LIN {X 0,Y 390.078,Z 257.397,A -85,B 0,C 180,E1 -11718.916,E2 -11718.916} C_VEL
LIN {X 0,Y 390.01,Z 257.402,A -85,B 0,C 180,E1 -11722.228,E2 -11722.228} C_VEL
LIN {X 0,Y 390.089,Z 257.39,A -85,B 0,C 180,E1 -11725.737,E2 -11725.737} C_VEL
LIN {X 0,Y 390.02,Z 257.4,A -85,B 0,C 180,E1 -11729.104,E2 -11729.104} C_VEL
LIN {X 0,Y 390.006,Z 257.404,A -85,B 0,C 180,E1 -11732.716,E2 -11732.716} C_VEL
LIN {X 0,Y 390.018,Z 257.4,A -85,B 0,C 180,E1 -11735.819,E2 -11735.819} C_VEL
LIN {X 0,Y 390.032,Z 257.397,A -85,B 0,C 180,E1 -11739.213,E2 -11739.213} C_VEL
LIN {X 0,Y 390.078,Z 257.396,A -85,B 0,C 180,E1 -11742.381,E2 -11742.381} C_VEL
LIN {X 0,Y 390.074,Z 257.392,A -85,B 0,C 180,E1 -11745.36,E2 -11745.36} C_VEL
LIN {X 0,Y 390.056,Z 257.399,A -85,B 0,C 180,E1 -11748.191,E2 -11748.191} C_VEL
LIN {X 0,Y 390.045,Z 257.396,A -85,B 0,C 180,E1 -11750.903,E2 -11750.903} C_VEL
LIN {X 0,Y 390.032,Z 257.397,A -85,B 0,C 180,E1 -11754.789,E2 -11754.789} C_VEL
LIN {X 0,Y 389.97,Z 257.405,A -85,B 0,C 180,E1 -11758.492,E2 -11758.492} C_VEL
LIN {X 0,Y 390.061,Z 257.396,A -85,B 0,C 180,E1 -11762.066,E2 -11762.066} C_VEL
LIN {X 0,Y 390.027,Z 257.404,A -85,B 0,C 180,E1 -11765.516,E2 -11765.516} C_VEL
LIN {X 0,Y 390.049,Z 257.396,A -85,B 0,C 180,E1 -11768.878,E2 -11768.878} C_VEL
LIN {X 0,Y 390.088,Z 257.395,A -85,B 0,C 180,E1 -11772.689,E2 -11772.689} C_VEL
LIN {X 0,Y 390.132,Z 257.39,A -85,B 0,C 180,E1 -11776.56,E2 -11776.56} C_VEL
LIN {X 0,Y 390.118,Z 257.391,A -85,B 0,C 180,E1 -11779.622,E2 -11779.622} C_VEL
LIN {X 0,Y 390.303,Z 257.447,A -85,B 0,C 180,E1 -11782.673,E2 -11782.673} C_VEL
LIN {X 0,Y 390.823,Z 259.339,A -85,B 0,C 180,E1 -11783.093,E2 -11783.093} C_VEL
LIN {X 0,Y 392.36,Z 261.617,A -85,B 0,C 180,E1 -11784.217,E2 -11784.217} C_VEL
LIN {X 0,Y 394.306,Z 263.039,A -85,B 0,C 180,E1 -11785.912,E2 -11785.912} C_VEL
LIN {X 0,Y 395.192,Z 263.267,A -85,B 0,C 180,E1 -11786.942,E2 -11786.942} C_VEL
LIN {X 0,Y 396.203,Z 263.5,A -85,B 0,C 180,E1 -11788.984,E2 -11788.984} C_VEL
LIN {X 0,Y 396.371,Z 263.477,A -85,B 0,C 180,E1 -11790,E2 -11790} C_VEL
LIN {X 0,Y 395.805,Z 263.406,A -85,B 0,C 180,E1 -11792.035,E2 -11792.035} C_VEL
LIN {X 0,Y 394.435,Z 263.067,A -85,B 0,C 180,E1 -11793.94,E2 -11793.94} C_VEL
LIN {X 0,Y 392.534,Z 261.798,A -85,B 0,C 180,E1 -11795.651,E2 -11795.651} C_VEL
LIN {X 0,Y 390.904,Z 259.538,A -85,B 0,C 180,E1 -11796.841,E2 -11796.841} C_VEL
LIN {X 0,Y 390.334,Z 257.663,A -85,B 0,C 180,E1 -11797.298,E2 -11797.298} C_VEL
LIN {X 0,Y 390.276,Z 257.373,A -85,B 0,C 180,E1 -11797.472,E2 -11797.472} C_VEL
LIN {X 0,Y 390.097,Z 257.393,A -85,B 0,C 180,E1 -11801.43,E2 -11801.43} C_VEL
LIN {X 0,Y 390.089,Z 257.397,A -85,B 0,C 180,E1 -11804.609,E2 -11804.609} C_VEL
LIN {X 0,Y 390.07,Z 257.397,A -85,B 0,C 180,E1 -11807.836,E2 -11807.836} C_VEL
LIN {X 0,Y 390.049,Z 257.396,A -85,B 0,C 180,E1 -11811.122,E2 -11811.122} C_VEL
LIN {X 0,Y 390.027,Z 257.404,A -85,B 0,C 180,E1 -11814.484,E2 -11814.484} C_VEL
LIN {X 0,Y 390.059,Z 257.397,A -85,B 0,C 180,E1 -11818.029,E2 -11818.029} C_VEL
LIN {X 0,Y 389.96,Z 257.408,A -85,B 0,C 180,E1 -11820.785,E2 -11820.785} C_VEL
LIN {X 0,Y 389.284,Z 257.493,A -85,B 0,C 180,E1 -11821.647,E2 -11821.647} C_VEL
LIN {X 0,Y 386.437,Z 257.845,A -85,B 0,C 180,E1 -11823.049,E2 -11823.049} C_VEL
LIN {X 0,Y 384.041,Z 258.15,A -85,B 0,C 180,E1 -11824.182,E2 -11824.182} C_VEL
LIN {X 0,Y 383.023,Z 258.271,A -85,B 0,C 180,E1 -11825.058,E2 -11825.058} C_VEL
LIN {X 0,Y 382.945,Z 258.28,A -85,B 0,C 180,E1 -11825.355,E2 -11825.355} C_VEL
LIN {X 0,Y 382.958,Z 258.28,A -85,B 0,C 180,E1 -11828.605,E2 -11828.605} C_VEL
LIN {X 0,Y 382.998,Z 258.274,A -85,B 0,C 180,E1 -11831.344,E2 -11831.344} C_VEL
LIN {X 0,Y 383.025,Z 258.272,A -85,B 0,C 180,E1 -11834.32,E2 -11834.32} C_VEL
LIN {X 0,Y 383.032,Z 258.271,A -85,B 0,C 180,E1 -11837.255,E2 -11837.255} C_VEL
LIN {X 0,Y 382.98,Z 258.276,A -85,B 0,C 180,E1 -11840.418,E2 -11840.418} C_VEL
LIN {X 0,Y 382.987,Z 258.277,A -85,B 0,C 180,E1 -11844.051,E2 -11844.051} C_VEL
LIN {X 0,Y 382.968,Z 258.284,A -85,B 0,C 180,E1 -11847.58,E2 -11847.58} C_VEL
LIN {X 0,Y 382.955,Z 258.279,A -85,B 0,C 180,E1 -11850.306,E2 -11850.306} C_VEL
LIN {X 0,Y 383.05,Z 258.268,A -85,B 0,C 180,E1 -11854.027,E2 -11854.027} C_VEL
LIN {X 0,Y 382.964,Z 258.284,A -85,B 0,C 180,E1 -11857.341,E2 -11857.341} C_VEL
LIN {X 0,Y 383.033,Z 258.271,A -85,B 0,C 180,E1 -11860.723,E2 -11860.723} C_VEL
LIN {X 0,Y 383.058,Z 258.266,A -85,B 0,C 180,E1 -11864.033,E2 -11864.033} C_VEL
LIN {X 0,Y 383.117,Z 258.263,A -85,B 0,C 180,E1 -11867.29,E2 -11867.29} C_VEL
LIN {X 0,Y 383.126,Z 258.259,A -85,B 0,C 180,E1 -11870.504,E2 -11870.504} C_VEL
LIN {X 0,Y 383.246,Z 258.243,A -85,B 0,C 180,E1 -11873.69,E2 -11873.69} C_VEL
LIN {X 0,Y 383.373,Z 258.227,A -85,B 0,C 180,E1 -11877.905,E2 -11877.905} C_VEL
LIN {X 0,Y 383.505,Z 258.211,A -85,B 0,C 180,E1 -11880.006,E2 -11880.006} C_VEL
LIN {X 0,Y 383.196,Z 258.251,A -85,B 0,C 180,E1 -11883.16,E2 -11883.16} C_VEL
LIN {X 0,Y 383.254,Z 258.245,A -85,B 0,C 180,E1 -11886.323,E2 -11886.323} C_VEL
LIN {X 0,Y 383.138,Z 258.256,A -85,B 0,C 180,E1 -11889.508,E2 -11889.508} C_VEL
LIN {X 0,Y 383.125,Z 258.258,A -85,B 0,C 180,E1 -11893.541,E2 -11893.541} C_VEL
LIN {X 0,Y 383.095,Z 258.262,A -85,B 0,C 180,E1 -11897.074,E2 -11897.074} C_VEL
LIN {X 0,Y 383.032,Z 258.272,A -85,B 0,C 180,E1 -11900.651,E2 -11900.651} C_VEL
LIN {X 0,Y 383.018,Z 258.274,A -85,B 0,C 180,E1 -11903.813,E2 -11903.813} C_VEL
LIN {X 0,Y 382.993,Z 258.274,A -85,B 0,C 180,E1 -11907.312,E2 -11907.312} C_VEL
LIN {X 0,Y 382.988,Z 258.275,A -85,B 0,C 180,E1 -11910.923,E2 -11910.923} C_VEL
LIN {X 0,Y 383.02,Z 258.274,A -85,B 0,C 180,E1 -11914.673,E2 -11914.673} C_VEL
LIN {X 0,Y 383.006,Z 258.279,A -85,B 0,C 180,E1 -11917.907,E2 -11917.907} C_VEL
LIN {X 0,Y 383.421,Z 261.152,A -85,B 0,C 180,E1 -11921.295,E2 -11921.295} C_VEL
LIN {X 0,Y 383.824,Z 264.04,A -85,B 0,C 180,E1 -11924.431,E2 -11924.431} C_VEL
LIN {X 0,Y 384.033,Z 267.009,A -85,B 0,C 180,E1 -11927.382,E2 -11927.382} C_VEL
LIN {X 0,Y 383.857,Z 270.176,A -85,B 0,C 180,E1 -11930.267,E2 -11930.267} C_VEL
LIN {X 0,Y 383.506,Z 274.24,A -85,B 0,C 180,E1 -11933.744,E2 -11933.744} C_VEL
LIN {X 0,Y 383.169,Z 277.795,A -85,B 0,C 180,E1 -11936.617,E2 -11936.617} C_VEL
LIN {X 0,Y 382.7,Z 282.543,A -85,B 0,C 180,E1 -11940.276,E2 -11940.276} C_VEL
LIN {X 0,Y 382.294,Z 287.36,A -85,B 0,C 180,E1 -11943.82,E2 -11943.82} C_VEL
LIN {X 0,Y 382.041,Z 292.216,A -85,B 0,C 180,E1 -11947.275,E2 -11947.275} C_VEL
LIN {X 0,Y 381.798,Z 297.479,A -85,B 0,C 180,E1 -11950.93,E2 -11950.93} C_VEL
LIN {X 0,Y 381.775,Z 297.832,A -85,B 0,C 180,E1 -11951.103,E2 -11951.103} C_VEL
LIN {X 0,Y 383.933,Z 308.212,A -85,B 0,C 180,E1 -11951.559,E2 -11951.559} C_VEL
LIN {X 0,Y 385.499,Z 317.173,A -85,B 0,C 180,E1 -11952.051,E2 -11952.051} C_VEL
LIN {X 0,Y 386.76,Z 326.079,A -85,B 0,C 180,E1 -11952.634,E2 -11952.634} C_VEL
LIN {X 0,Y 387.065,Z 332.785,A -85,B 0,C 180,E1 -11953.112,E2 -11953.112} C_VEL
LIN {X 0,Y 386.15,Z 343.695,A -85,B 0,C 180,E1 -11954.022,E2 -11954.022} C_VEL
LIN {X 0,Y 385.323,Z 352.64,A -85,B 0,C 180,E1 -11954.936,E2 -11954.936} C_VEL
LIN {X 0,Y 384.651,Z 360.342,A -85,B 0,C 180,E1 -11955.874,E2 -11955.874} C_VEL
LIN {X 0,Y 383.975,Z 368.393,A -85,B 0,C 180,E1 -11957.044,E2 -11957.044} C_VEL
LIN {X 0,Y 383.342,Z 374.594,A -85,B 0,C 180,E1 -11958.098,E2 -11958.098} C_VEL
LIN {X 0,Y 382.751,Z 381.132,A -85,B 0,C 180,E1 -11959.42,E2 -11959.42} C_VEL
LIN {X 0,Y 382.377,Z 385.634,A -85,B 0,C 180,E1 -11960.479,E2 -11960.479} C_VEL
LIN {X 0,Y 381.964,Z 391.125,A -85,B 0,C 180,E1 -11962.068,E2 -11962.068} C_VEL
LIN {X 0,Y 381.726,Z 395.45,A -85,B 0,C 180,E1 -11963.658,E2 -11963.658} C_VEL
LIN {X 0,Y 381.65,Z 397.817,A -85,B 0,C 180,E1 -11964.717,E2 -11964.717} C_VEL
LIN {X 0,Y 381.624,Z 399.616,A -85,B 0,C 180,E1 -11965.776,E2 -11965.776} C_VEL
LIN {X 0,Y 381.563,Z 402.06,A -85,B 0,C 180,E1 -11967.889,E2 -11967.889} C_VEL
LIN {X 0,Y 381.598,Z 402.649,A -85,B 0,C 180,E1 -11968.945,E2 -11968.945} C_VEL
LIN {X 0,Y 381.598,Z 402.649,A -85,B 0,C 180,E1 -11971.055,E2 -11971.055} C_VEL
LIN {X 0,Y 381.563,Z 402.06,A -85,B 0,C 180,E1 -11972.111,E2 -11972.111} C_VEL
LIN {X 0,Y 381.624,Z 399.616,A -85,B 0,C 180,E1 -11974.224,E2 -11974.224} C_VEL
LIN {X 0,Y 381.65,Z 397.817,A -85,B 0,C 180,E1 -11975.283,E2 -11975.283} C_VEL
LIN {X 0,Y 381.795,Z 394.21,A -85,B 0,C 180,E1 -11976.872,E2 -11976.872} C_VEL
LIN {X 0,Y 382.075,Z 389.465,A -85,B 0,C 180,E1 -11978.462,E2 -11978.462} C_VEL
LIN {X 0,Y 382.544,Z 383.443,A -85,B 0,C 180,E1 -11980.051,E2 -11980.051} C_VEL
LIN {X 0,Y 383.071,Z 377.346,A -85,B 0,C 180,E1 -11981.374,E2 -11981.374} C_VEL
LIN {X 0,Y 383.641,Z 371.646,A -85,B 0,C 180,E1 -11982.43,E2 -11982.43} C_VEL
LIN {X 0,Y 384.394,Z 363.091,A -85,B 0,C 180,E1 -11983.749,E2 -11983.749} C_VEL
LIN {X 0,Y 385.11,Z 354.909,A -85,B 0,C 180,E1 -11984.802,E2 -11984.802} C_VEL
LIN {X 0,Y 385.872,Z 346.398,A -85,B 0,C 180,E1 -11985.719,E2 -11985.719} C_VEL
LIN {X 0,Y 386.581,Z 337.681,A -85,B 0,C 180,E1 -11986.502,E2 -11986.502} C_VEL
LIN {X 0,Y 387.137,Z 330.218,A -85,B 0,C 180,E1 -11987.07,E2 -11987.07} C_VEL
LIN {X 0,Y 386.004,Z 320.346,A -85,B 0,C 180,E1 -11987.757,E2 -11987.757} C_VEL
LIN {X 0,Y 384.122,Z 309.199,A -85,B 0,C 180,E1 -11988.392,E2 -11988.392} C_VEL
LIN {X 0,Y 381.847,Z 298.335,A -85,B 0,C 180,E1 -11988.88,E2 -11988.88} C_VEL
LIN {X 0,Y 381.777,Z 297.67,A -85,B 0,C 180,E1 -11988.932,E2 -11988.932} C_VEL
LIN {X 0,Y 382.043,Z 292.21,A -85,B 0,C 180,E1 -11992.725,E2 -11992.725} C_VEL
LIN {X 0,Y 382.294,Z 287.352,A -85,B 0,C 180,E1 -11996.18,E2 -11996.18} C_VEL
LIN {X 0,Y 382.701,Z 282.543,A -85,B 0,C 180,E1 -11999.724,E2 -11999.724} C_VEL
LIN {X 0,Y 383.07,Z 278.991,A -85,B 0,C 180,E1 -12002.436,E2 -12002.436} C_VEL
LIN {X 0,Y 383.457,Z 274.66,A -85,B 0,C 180,E1 -12005.908,E2 -12005.908} C_VEL
LIN {X 0,Y 383.718,Z 271.563,A -85,B 0,C 180,E1 -12008.514,E2 -12008.514} C_VEL
LIN {X 0,Y 383.974,Z 268.349,A -85,B 0,C 180,E1 -12011.367,E2 -12011.367} C_VEL
LIN {X 0,Y 383.99,Z 265.506,A -85,B 0,C 180,E1 -12014.066,E2 -12014.066} C_VEL
LIN {X 0,Y 383.565,Z 262.396,A -85,B 0,C 180,E1 -12017.312,E2 -12017.312} C_VEL
LIN {X 0,Y 383.222,Z 259.706,A -85,B 0,C 180,E1 -12020.374,E2 -12020.374} C_VEL
LIN {X 0,Y 383.007,Z 258.279,A -85,B 0,C 180,E1 -12022.093,E2 -12022.093} C_VEL
LIN {X 0,Y 383.025,Z 258.277,A -85,B 0,C 180,E1 -12025.328,E2 -12025.328} C_VEL
LIN {X 0,Y 382.988,Z 258.275,A -85,B 0,C 180,E1 -12029.077,E2 -12029.077} C_VEL
LIN {X 0,Y 382.993,Z 258.274,A -85,B 0,C 180,E1 -12032.688,E2 -12032.688} C_VEL
LIN {X 0,Y 383.018,Z 258.274,A -85,B 0,C 180,E1 -12036.187,E2 -12036.187} C_VEL
LIN {X 0,Y 383.058,Z 258.271,A -85,B 0,C 180,E1 -12039.593,E2 -12039.593} C_VEL
LIN {X 0,Y 383.095,Z 258.262,A -85,B 0,C 180,E1 -12042.926,E2 -12042.926} C_VEL
LIN {X 0,Y 383.125,Z 258.258,A -85,B 0,C 180,E1 -12046.459,E2 -12046.459} C_VEL
LIN {X 0,Y 383.138,Z 258.256,A -85,B 0,C 180,E1 -12050.492,E2 -12050.492} C_VEL
LIN {X 0,Y 383.254,Z 258.245,A -85,B 0,C 180,E1 -12053.677,E2 -12053.677} C_VEL
LIN {X 0,Y 383.366,Z 258.229,A -85,B 0,C 180,E1 -12057.893,E2 -12057.893} C_VEL
LIN {X 0,Y 383.505,Z 258.211,A -85,B 0,C 180,E1 -12059.994,E2 -12059.994} C_VEL
LIN {X 0,Y 383.23,Z 258.251,A -85,B 0,C 180,E1 -12063.147,E2 -12063.147} C_VEL
LIN {X 0,Y 383.225,Z 258.245,A -85,B 0,C 180,E1 -12066.59,E2 -12066.59} C_VEL
LIN {X 0,Y 383.126,Z 258.259,A -85,B 0,C 180,E1 -12069.496,E2 -12069.496} C_VEL
LIN {X 0,Y 383.106,Z 258.261,A -85,B 0,C 180,E1 -12073.53,E2 -12073.53} C_VEL
LIN {X 0,Y 383.071,Z 258.268,A -85,B 0,C 180,E1 -12077.063,E2 -12077.063} C_VEL
LIN {X 0,Y 383.003,Z 258.279,A -85,B 0,C 180,E1 -12080.64,E2 -12080.64} C_VEL
LIN {X 0,Y 382.994,Z 258.274,A -85,B 0,C 180,E1 -12083.802,E2 -12083.802} C_VEL
LIN {X 0,Y 383.049,Z 258.269,A -85,B 0,C 180,E1 -12086.117,E2 -12086.117} C_VEL
LIN {X 0,Y 382.955,Z 258.279,A -85,B 0,C 180,E1 -12089.694,E2 -12089.694} C_VEL
LIN {X 0,Y 382.966,Z 258.277,A -85,B 0,C 180,E1 -12093.395,E2 -12093.395} C_VEL
LIN {X 0,Y 382.994,Z 258.279,A -85,B 0,C 180,E1 -12096.159,E2 -12096.159} C_VEL
LIN {X 0,Y 382.978,Z 258.279,A -85,B 0,C 180,E1 -12099.951,E2 -12099.951} C_VEL
LIN {X 0,Y 383.022,Z 258.272,A -85,B 0,C 180,E1 -12102.783,E2 -12102.783} C_VEL
LIN {X 0,Y 383.027,Z 258.273,A -85,B 0,C 180,E1 -12105.795,E2 -12105.795} C_VEL
LIN {X 0,Y 382.996,Z 258.274,A -85,B 0,C 180,E1 -12108.781,E2 -12108.781} C_VEL
LIN {X 0,Y 382.952,Z 258.284,A -85,B 0,C 180,E1 -12112.091,E2 -12112.091} C_VEL
LIN {X 0,Y 382.965,Z 258.279,A -85,B 0,C 180,E1 -12115.328,E2 -12115.328} C_VEL
LIN {X 0,Y 382.93,Z 258.283,A -85,B 0,C 180,E1 -12119.078,E2 -12119.078} C_VEL
LIN {X 0,Y 382.999,Z 258.273,A -85,B 0,C 180,E1 -12122.694,E2 -12122.694} C_VEL
LIN {X 0,Y 382.99,Z 258.276,A -85,B 0,C 180,E1 -12126.19,E2 -12126.19} C_VEL
LIN {X 0,Y 383.022,Z 258.277,A -85,B 0,C 180,E1 -12129.597,E2 -12129.597} C_VEL
LIN {X 0,Y 383.045,Z 258.273,A -85,B 0,C 180,E1 -12132.929,E2 -12132.929} C_VEL
LIN {X 0,Y 383.063,Z 258.27,A -85,B 0,C 180,E1 -12136.462,E2 -12136.462} C_VEL
LIN {X 0,Y 383.112,Z 258.454,A -85,B 0,C 180,E1 -12139.597,E2 -12139.597} C_VEL
LIN {X 0,Y 383.731,Z 260.437,A -85,B 0,C 180,E1 -12139.914,E2 -12139.914} C_VEL
LIN {X 0,Y 385.194,Z 262.473,A -85,B 0,C 180,E1 -12140.615,E2 -12140.615} C_VEL
LIN {X 0,Y 387.433,Z 263.895,A -85,B 0,C 180,E1 -12141.656,E2 -12141.656} C_VEL
LIN {X 0,Y 388.819,Z 264.578,A -85,B 0,C 180,E1 -12142.393,E2 -12142.393} C_VEL
LIN {X 0,Y 389.954,Z 266.887,A -85,B 0,C 180,E1 -12143.142,E2 -12143.142} C_VEL
LIN {X 0,Y 391.787,Z 269.021,A -85,B 0,C 180,E1 -12144.467,E2 -12144.467} C_VEL
LIN {X 0,Y 393.419,Z 270.082,A -85,B 0,C 180,E1 -12145.903,E2 -12145.903} C_VEL
LIN {X 0,Y 394.315,Z 270.311,A -85,B 0,C 180,E1 -12146.935,E2 -12146.935} C_VEL
LIN {X 0,Y 395.344,Z 270.547,A -85,B 0,C 180,E1 -12148.981,E2 -12148.981} C_VEL
LIN {X 0,Y 395.505,Z 270.523,A -85,B 0,C 180,E1 -12150,E2 -12150} C_VEL
LIN {X 0,Y 394.942,Z 270.452,A -85,B 0,C 180,E1 -12152.04,E2 -12152.04} C_VEL
LIN {X 0,Y 393.419,Z 270.083,A -85,B 0,C 180,E1 -12154.097,E2 -12154.097} C_VEL
LIN {X 0,Y 391.44,Z 268.741,A -85,B 0,C 180,E1 -12155.796,E2 -12155.796} C_VEL
LIN {X 0,Y 389.612,Z 266.328,A -85,B 0,C 180,E1 -12157.089,E2 -12157.089} C_VEL
LIN {X 0,Y 388.598,Z 264.268,A -85,B 0,C 180,E1 -12157.735,E2 -12157.735} C_VEL
LIN {X 0,Y 386.111,Z 263.175,A -85,B 0,C 180,E1 -12158.966,E2 -12158.966} C_VEL
LIN {X 0,Y 384.201,Z 261.296,A -85,B 0,C 180,E1 -12159.861,E2 -12159.861} C_VEL
LIN {X 0,Y 383.293,Z 259.34,A -85,B 0,C 180,E1 -12160.298,E2 -12160.298} C_VEL
LIN {X 0,Y 383.073,Z 258.269,A -85,B 0,C 180,E1 -12160.438,E2 -12160.438} C_VEL
LIN {X 0,Y 383.066,Z 258.269,A -85,B 0,C 180,E1 -12163.798,E2 -12163.798} C_VEL
LIN {X 0,Y 383.035,Z 258.273,A -85,B 0,C 180,E1 -12167.458,E2 -12167.458} C_VEL
LIN {X 0,Y 383.004,Z 258.277,A -85,B 0,C 180,E1 -12170.664,E2 -12170.664} C_VEL
LIN {X 0,Y 382.99,Z 258.276,A -85,B 0,C 180,E1 -12173.81,E2 -12173.81} C_VEL
LIN {X 0,Y 382.999,Z 258.273,A -85,B 0,C 180,E1 -12177.306,E2 -12177.306} C_VEL
LIN {X 0,Y 382.93,Z 258.283,A -85,B 0,C 180,E1 -12180.922,E2 -12180.922} C_VEL
LIN {X 0,Y 382.965,Z 258.279,A -85,B 0,C 180,E1 -12184.672,E2 -12184.672} C_VEL
LIN {X 0,Y 382.945,Z 258.28,A -85,B 0,C 180,E1 -12185.355,E2 -12185.355} C_VEL
LIN {X 0,Y 382.302,Z 258.366,A -85,B 0,C 180,E1 -12186.233,E2 -12186.233} C_VEL
LIN {X 0,Y 379.489,Z 258.724,A -85,B 0,C 180,E1 -12187.661,E2 -12187.661} C_VEL
LIN {X 0,Y 377.087,Z 259.025,A -85,B 0,C 180,E1 -12188.816,E2 -12188.816} C_VEL
LIN {X 0,Y 376.041,Z 259.149,A -85,B 0,C 180,E1 -12189.708,E2 -12189.708} C_VEL
LIN {X 0,Y 375.949,Z 259.158,A -85,B 0,C 180,E1 -12190.01,E2 -12190.01} C_VEL
LIN {X 0,Y 375.955,Z 259.156,A -85,B 0,C 180,E1 -12193.761,E2 -12193.761} C_VEL
LIN {X 0,Y 375.955,Z 259.151,A -85,B 0,C 180,E1 -12196.806,E2 -12196.806} C_VEL
LIN {X 0,Y 375.957,Z 259.154,A -85,B 0,C 180,E1 -12200.034,E2 -12200.034} C_VEL
LIN {X 0,Y 375.926,Z 259.159,A -85,B 0,C 180,E1 -12203.501,E2 -12203.501} C_VEL
LIN {X 0,Y 375.923,Z 259.158,A -85,B 0,C 180,E1 -12205.895,E2 -12205.895} C_VEL
LIN {X 0,Y 375.929,Z 259.159,A -85,B 0,C 180,E1 -12209.694,E2 -12209.694} C_VEL
LIN {X 0,Y 375.989,Z 259.152,A -85,B 0,C 180,E1 -12213.354,E2 -12213.354} C_VEL
LIN {X 0,Y 375.951,Z 259.153,A -85,B 0,C 180,E1 -12216.894,E2 -12216.894} C_VEL
LIN {X 0,Y 375.971,Z 259.149,A -85,B 0,C 180,E1 -12220.346,E2 -12220.346} C_VEL
LIN {X 0,Y 376.003,Z 259.146,A -85,B 0,C 180,E1 -12223.725,E2 -12223.725} C_VEL
LIN {X 0,Y 376.084,Z 259.141,A -85,B 0,C 180,E1 -12227.049,E2 -12227.049} C_VEL
LIN {X 0,Y 376.096,Z 259.134,A -85,B 0,C 180,E1 -12230.325,E2 -12230.325} C_VEL
LIN {X 0,Y 376.205,Z 259.121,A -85,B 0,C 180,E1 -12233.571,E2 -12233.571} C_VEL
LIN {X 0,Y 376.339,Z 259.103,A -85,B 0,C 180,E1 -12237.866,E2 -12237.866} C_VEL
LIN {X 0,Y 376.474,Z 259.086,A -85,B 0,C 180,E1 -12240.006,E2 -12240.006} C_VEL
LIN {X 0,Y 376.331,Z 259.105,A -85,B 0,C 180,E1 -12242.147,E2 -12242.147} C_VEL
LIN {X 0,Y 376.213,Z 259.123,A -85,B 0,C 180,E1 -12246.441,E2 -12246.441} C_VEL
LIN {X 0,Y 376.109,Z 259.132,A -85,B 0,C 180,E1 -12249.687,E2 -12249.687} C_VEL
LIN {X 0,Y 376.089,Z 259.134,A -85,B 0,C 180,E1 -12253.663,E2 -12253.663} C_VEL
LIN {X 0,Y 376.034,Z 259.141,A -85,B 0,C 180,E1 -12257.405,E2 -12257.405} C_VEL
LIN {X 0,Y 375.982,Z 259.149,A -85,B 0,C 180,E1 -12260.837,E2 -12260.837} C_VEL
LIN {X 0,Y 375.967,Z 259.154,A -85,B 0,C 180,E1 -12264.289,E2 -12264.289} C_VEL
LIN {X 0,Y 375.937,Z 259.157,A -85,B 0,C 180,E1 -12267.869,E2 -12267.869} C_VEL
LIN {X 0,Y 375.964,Z 259.152,A -85,B 0,C 180,E1 -12271.567,E2 -12271.567} C_VEL
LIN {X 0,Y 375.958,Z 259.153,A -85,B 0,C 180,E1 -12275.421,E2 -12275.421} C_VEL
LIN {X 0,Y 375.958,Z 259.155,A -85,B 0,C 180,E1 -12276.746,E2 -12276.746} C_VEL
LIN {X 0,Y 376.032,Z 259.734,A -85,B 0,C 180,E1 -12278.283,E2 -12278.283} C_VEL
LIN {X 0,Y 376.457,Z 262.579,A -85,B 0,C 180,E1 -12281.692,E2 -12281.692} C_VEL
LIN {X 0,Y 376.875,Z 265.757,A -85,B 0,C 180,E1 -12285.129,E2 -12285.129} C_VEL
LIN {X 0,Y 376.966,Z 268.497,A -85,B 0,C 180,E1 -12287.844,E2 -12287.844} C_VEL
LIN {X 0,Y 376.776,Z 271.531,A -85,B 0,C 180,E1 -12290.64,E2 -12290.64} C_VEL
LIN {X 0,Y 376.488,Z 274.693,A -85,B 0,C 180,E1 -12293.394,E2 -12293.394} C_VEL
LIN {X 0,Y 376.039,Z 279.289,A -85,B 0,C 180,E1 -12297.181,E2 -12297.181} C_VEL
LIN {X 0,Y 375.738,Z 282.45,A -85,B 0,C 180,E1 -12299.668,E2 -12299.668} C_VEL
LIN {X 0,Y 375.267,Z 287.244,A -85,B 0,C 180,E1 -12303.291,E2 -12303.291} C_VEL
LIN {X 0,Y 375.003,Z 292.076,A -85,B 0,C 180,E1 -12306.824,E2 -12306.824} C_VEL
LIN {X 0,Y 374.753,Z 297.629,A -85,B 0,C 180,E1 -12310.735,E2 -12310.735} C_VEL
LIN {X 0,Y 376.778,Z 307.363,A -85,B 0,C 180,E1 -12311.17,E2 -12311.17} C_VEL
LIN {X 0,Y 378.522,Z 317.005,A -85,B 0,C 180,E1 -12311.711,E2 -12311.711} C_VEL
LIN {X 0,Y 379.834,Z 326.248,A -85,B 0,C 180,E1 -12312.333,E2 -12312.333} C_VEL
LIN {X 0,Y 380.262,Z 332.59,A -85,B 0,C 180,E1 -12312.8,E2 -12312.8} C_VEL
LIN {X 0,Y 379.323,Z 343.5,A -85,B 0,C 180,E1 -12313.726,E2 -12313.726} C_VEL
LIN {X 0,Y 378.437,Z 352.444,A -85,B 0,C 180,E1 -12314.655,E2 -12314.655} C_VEL
LIN {X 0,Y 377.712,Z 360.515,A -85,B 0,C 180,E1 -12315.662,E2 -12315.662} C_VEL
LIN {X 0,Y 377.039,Z 368.198,A -85,B 0,C 180,E1 -12316.801,E2 -12316.801} C_VEL
LIN {X 0,Y 376.386,Z 374.399,A -85,B 0,C 180,E1 -12317.874,E2 -12317.874} C_VEL
LIN {X 0,Y 375.73,Z 380.936,A -85,B 0,C 180,E1 -12319.22,E2 -12319.22} C_VEL
LIN {X 0,Y 375.336,Z 385.438,A -85,B 0,C 180,E1 -12320.298,E2 -12320.298} C_VEL
LIN {X 0,Y 374.901,Z 390.93,A -85,B 0,C 180,E1 -12321.918,E2 -12321.918} C_VEL
LIN {X 0,Y 374.647,Z 395.255,A -85,B 0,C 180,E1 -12323.538,E2 -12323.538} C_VEL
LIN {X 0,Y 374.561,Z 397.622,A -85,B 0,C 180,E1 -12324.617,E2 -12324.617} C_VEL
LIN {X 0,Y 374.53,Z 399.421,A -85,B 0,C 180,E1 -12325.695,E2 -12325.695} C_VEL
LIN {X 0,Y 374.462,Z 401.865,A -85,B 0,C 180,E1 -12327.849,E2 -12327.849} C_VEL
LIN {X 0,Y 374.499,Z 402.455,A -85,B 0,C 180,E1 -12328.925,E2 -12328.925} C_VEL
LIN {X 0,Y 374.499,Z 402.455,A -85,B 0,C 180,E1 -12331.075,E2 -12331.075} C_VEL
LIN {X 0,Y 374.462,Z 401.865,A -85,B 0,C 180,E1 -12332.151,E2 -12332.151} C_VEL
LIN {X 0,Y 374.53,Z 399.421,A -85,B 0,C 180,E1 -12334.305,E2 -12334.305} C_VEL
LIN {X 0,Y 374.595,Z 396.162,A -85,B 0,C 180,E1 -12336.06,E2 -12336.06} C_VEL
LIN {X 0,Y 374.812,Z 392.484,A -85,B 0,C 180,E1 -12337.542,E2 -12337.542} C_VEL
LIN {X 0,Y 375.175,Z 387.354,A -85,B 0,C 180,E1 -12339.162,E2 -12339.162} C_VEL
LIN {X 0,Y 375.65,Z 382.092,A -85,B 0,C 180,E1 -12340.51,E2 -12340.51} C_VEL
LIN {X 0,Y 376.217,Z 375.774,A -85,B 0,C 180,E1 -12341.858,E2 -12341.858} C_VEL
LIN {X 0,Y 376.877,Z 369.825,A -85,B 0,C 180,E1 -12342.931,E2 -12342.931} C_VEL
LIN {X 0,Y 377.62,Z 361.709,A -85,B 0,C 180,E1 -12344.171,E2 -12344.171} C_VEL
LIN {X 0,Y 378.421,Z 352.443,A -85,B 0,C 180,E1 -12345.346,E2 -12345.346} C_VEL
LIN {X 0,Y 379.385,Z 342.147,A -85,B 0,C 180,E1 -12346.409,E2 -12346.409} C_VEL
LIN {X 0,Y 380.288,Z 331.449,A -85,B 0,C 180,E1 -12347.288,E2 -12347.288} C_VEL
LIN {X 0,Y 379.081,Z 320.707,A -85,B 0,C 180,E1 -12348.062,E2 -12348.062} C_VEL
LIN {X 0,Y 377.189,Z 309.445,A -85,B 0,C 180,E1 -12348.725,E2 -12348.725} C_VEL
LIN {X 0,Y 374.81,Z 298.298,A -85,B 0,C 180,E1 -12349.244,E2 -12349.244} C_VEL
LIN {X 0,Y 374.752,Z 297.506,A -85,B 0,C 180,E1 -12349.3,E2 -12349.3} C_VEL
LIN {X 0,Y 375.016,Z 291.876,A -85,B 0,C 180,E1 -12353.316,E2 -12353.316} C_VEL
LIN {X 0,Y 375.266,Z 287.234,A -85,B 0,C 180,E1 -12356.709,E2 -12356.709} C_VEL
LIN {X 0,Y 375.763,Z 282.052,A -85,B 0,C 180,E1 -12360.638,E2 -12360.638} C_VEL
LIN {X 0,Y 376.182,Z 277.711,A -85,B 0,C 180,E1 -12364.088,E2 -12364.088} C_VEL
LIN {X 0,Y 376.494,Z 274.604,A -85,B 0,C 180,E1 -12366.679,E2 -12366.679} C_VEL
LIN {X 0,Y 376.831,Z 270.678,A -85,B 0,C 180,E1 -12370.118,E2 -12370.118} C_VEL
LIN {X 0,Y 377.005,Z 267.25,A -85,B 0,C 180,E1 -12373.357,E2 -12373.357} C_VEL
LIN {X 0,Y 376.648,Z 264.045,A -85,B 0,C 180,E1 -12376.694,E2 -12376.694} C_VEL
LIN {X 0,Y 376.183,Z 260.68,A -85,B 0,C 180,E1 -12380.56,E2 -12380.56} C_VEL
LIN {X 0,Y 376.014,Z 259.579,A -85,B 0,C 180,E1 -12381.912,E2 -12381.912} C_VEL
LIN {X 0,Y 375.971,Z 259.154,A -85,B 0,C 180,E1 -12383.492,E2 -12383.492} C_VEL
LIN {X 0,Y 375.967,Z 259.156,A -85,B 0,C 180,E1 -12385.884,E2 -12385.884} C_VEL
LIN {X 0,Y 375.969,Z 259.152,A -85,B 0,C 180,E1 -12389.683,E2 -12389.683} C_VEL
LIN {X 0,Y 375.937,Z 259.157,A -85,B 0,C 180,E1 -12392.131,E2 -12392.131} C_VEL
LIN {X 0,Y 375.967,Z 259.154,A -85,B 0,C 180,E1 -12395.711,E2 -12395.711} C_VEL
LIN {X 0,Y 375.983,Z 259.149,A -85,B 0,C 180,E1 -12399.192,E2 -12399.192} C_VEL
LIN {X 0,Y 376.034,Z 259.141,A -85,B 0,C 180,E1 -12402.595,E2 -12402.595} C_VEL
LIN {X 0,Y 376.089,Z 259.134,A -85,B 0,C 180,E1 -12406.337,E2 -12406.337} C_VEL
LIN {X 0,Y 376.109,Z 259.132,A -85,B 0,C 180,E1 -12410.313,E2 -12410.313} C_VEL
LIN {X 0,Y 376.213,Z 259.123,A -85,B 0,C 180,E1 -12413.559,E2 -12413.559} C_VEL
LIN {X 0,Y 376.331,Z 259.105,A -85,B 0,C 180,E1 -12417.853,E2 -12417.853} C_VEL
LIN {X 0,Y 376.474,Z 259.086,A -85,B 0,C 180,E1 -12419.994,E2 -12419.994} C_VEL
LIN {X 0,Y 376.339,Z 259.103,A -85,B 0,C 180,E1 -12422.134,E2 -12422.134} C_VEL
LIN {X 0,Y 376.191,Z 259.121,A -85,B 0,C 180,E1 -12426.577,E2 -12426.577} C_VEL
LIN {X 0,Y 376.096,Z 259.134,A -85,B 0,C 180,E1 -12429.675,E2 -12429.675} C_VEL
LIN {X 0,Y 376.07,Z 259.137,A -85,B 0,C 180,E1 -12433.651,E2 -12433.651} C_VEL
LIN {X 0,Y 376.009,Z 259.145,A -85,B 0,C 180,E1 -12437.393,E2 -12437.393} C_VEL
LIN {X 0,Y 375.953,Z 259.156,A -85,B 0,C 180,E1 -12440.826,E2 -12440.826} C_VEL
LIN {X 0,Y 375.959,Z 259.153,A -85,B 0,C 180,E1 -12444.275,E2 -12444.275} C_VEL
LIN {X 0,Y 375.989,Z 259.152,A -85,B 0,C 180,E1 -12446.646,E2 -12446.646} C_VEL
LIN {X 0,Y 375.929,Z 259.159,A -85,B 0,C 180,E1 -12450.306,E2 -12450.306} C_VEL
LIN {X 0,Y 375.923,Z 259.158,A -85,B 0,C 180,E1 -12454.105,E2 -12454.105} C_VEL
LIN {X 0,Y 375.916,Z 259.158,A -85,B 0,C 180,E1 -12456.735,E2 -12456.735} C_VEL
LIN {X 0,Y 375.957,Z 259.154,A -85,B 0,C 180,E1 -12459.966,E2 -12459.966} C_VEL
LIN {X 0,Y 375.955,Z 259.151,A -85,B 0,C 180,E1 -12463.194,E2 -12463.194} C_VEL
LIN {X 0,Y 375.955,Z 259.156,A -85,B 0,C 180,E1 -12466.239,E2 -12466.239} C_VEL
LIN {X 0,Y 375.95,Z 259.158,A -85,B 0,C 180,E1 -12470.022,E2 -12470.022} C_VEL
LIN {X 0,Y 375.913,Z 259.158,A -85,B 0,C 180,E1 -12473.491,E2 -12473.491} C_VEL
LIN {X 0,Y 375.907,Z 259.163,A -85,B 0,C 180,E1 -12475.884,E2 -12475.884} C_VEL
LIN {X 0,Y 375.912,Z 259.162,A -85,B 0,C 180,E1 -12479.684,E2 -12479.684} C_VEL
LIN {X 0,Y 375.945,Z 259.154,A -85,B 0,C 180,E1 -12482.138,E2 -12482.138} C_VEL
LIN {X 0,Y 375.949,Z 259.152,A -85,B 0,C 180,E1 -12484.536,E2 -12484.536} C_VEL
LIN {X 0,Y 375.965,Z 259.151,A -85,B 0,C 180,E1 -12488.046,E2 -12488.046} C_VEL
LIN {X 0,Y 375.971,Z 259.155,A -85,B 0,C 180,E1 -12491.472,E2 -12491.472} C_VEL
LIN {X 0,Y 376.002,Z 259.151,A -85,B 0,C 180,E1 -12494.831,E2 -12494.831} C_VEL
LIN {X 0,Y 376.055,Z 259.145,A -85,B 0,C 180,E1 -12497.281,E2 -12497.281} C_VEL
LIN {X 0,Y 376.677,Z 261.346,A -85,B 0,C 180,E1 -12497.576,E2 -12497.576} C_VEL
LIN {X 0,Y 378.172,Z 263.406,A -85,B 0,C 180,E1 -12498.136,E2 -12498.136} C_VEL
LIN {X 0,Y 380.472,Z 264.884,A -85,B 0,C 180,E1 -12498.951,E2 -12498.951} C_VEL
LIN {X 0,Y 381.114,Z 265.313,A -85,B 0,C 180,E1 -12499.206,E2 -12499.206} C_VEL
LIN {X 0,Y 382.557,Z 267.93,A -85,B 0,C 180,E1 -12499.849,E2 -12499.849} C_VEL
LIN {X 0,Y 384.826,Z 270.07,A -85,B 0,C 180,E1 -12500.871,E2 -12500.871} C_VEL
LIN {X 0,Y 387.387,Z 271.481,A -85,B 0,C 180,E1 -12502.118,E2 -12502.118} C_VEL
LIN {X 0,Y 389.029,Z 274.175,A -85,B 0,C 180,E1 -12503.143,E2 -12503.143} C_VEL
LIN {X 0,Y 390.886,Z 276.104,A -85,B 0,C 180,E1 -12504.454,E2 -12504.454} C_VEL
LIN {X 0,Y 392.53,Z 277.125,A -85,B 0,C 180,E1 -12505.893,E2 -12505.893} C_VEL
LIN {X 0,Y 394.08,Z 277.499,A -85,B 0,C 180,E1 -12507.956,E2 -12507.956} C_VEL
LIN {X 0,Y 394.642,Z 277.556,A -85,B 0,C 180,E1 -12510,E2 -12510} C_VEL
LIN {X 0,Y 394.079,Z 277.498,A -85,B 0,C 180,E1 -12512.044,E2 -12512.044} C_VEL
LIN {X 0,Y 392.53,Z 277.126,A -85,B 0,C 180,E1 -12514.107,E2 -12514.107} C_VEL
LIN {X 0,Y 390.526,Z 275.82,A -85,B 0,C 180,E1 -12515.81,E2 -12515.81} C_VEL
LIN {X 0,Y 388.468,Z 273.382,A -85,B 0,C 180,E1 -12517.227,E2 -12517.227} C_VEL
LIN {X 0,Y 387.165,Z 271.164,A -85,B 0,C 180,E1 -12518.013,E2 -12518.013} C_VEL
LIN {X 0,Y 384.668,Z 269.991,A -85,B 0,C 180,E1 -12519.199,E2 -12519.199} C_VEL
LIN {X 0,Y 382.39,Z 267.719,A -85,B 0,C 180,E1 -12520.222,E2 -12520.222} C_VEL
LIN {X 0,Y 380.993,Z 265.034,A -85,B 0,C 180,E1 -12520.852,E2 -12520.852} C_VEL
LIN {X 0,Y 378.576,Z 263.788,A -85,B 0,C 180,E1 -12521.722,E2 -12521.722} C_VEL
LIN {X 0,Y 376.764,Z 261.561,A -85,B 0,C 180,E1 -12522.387,E2 -12522.387} C_VEL
LIN {X 0,Y 376.031,Z 259.148,A -85,B 0,C 180,E1 -12522.754,E2 -12522.754} C_VEL
LIN {X 0,Y 375.972,Z 259.154,A -85,B 0,C 180,E1 -12526.283,E2 -12526.283} C_VEL
LIN {X 0,Y 375.958,Z 259.155,A -85,B 0,C 180,E1 -12529.662,E2 -12529.662} C_VEL
LIN {X 0,Y 375.971,Z 259.149,A -85,B 0,C 180,E1 -12533.113,E2 -12533.113} C_VEL
LIN {X 0,Y 375.962,Z 259.153,A -85,B 0,C 180,E1 -12536.656,E2 -12536.656} C_VEL
LIN {X 0,Y 375.92,Z 259.155,A -85,B 0,C 180,E1 -12539.083,E2 -12539.083} C_VEL
LIN {X 0,Y 375.895,Z 259.159,A -85,B 0,C 180,E1 -12542.833,E2 -12542.833} C_VEL
LIN {X 0,Y 375.905,Z 259.158,A -85,B 0,C 180,E1 -12545.42,E2 -12545.42} C_VEL
LIN {X 0,Y 375.927,Z 259.158,A -85,B 0,C 180,E1 -12548.276,E2 -12548.276} C_VEL
LIN {X 0,Y 375.949,Z 259.158,A -85,B 0,C 180,E1 -12550.01,E2 -12550.01} C_VEL
LIN {X 0,Y 375.254,Z 259.238,A -85,B 0,C 180,E1 -12550.904,E2 -12550.904} C_VEL
LIN {X 0,Y 372.381,Z 259.598,A -85,B 0,C 180,E1 -12552.357,E2 -12552.357} C_VEL
LIN {X 0,Y 369.989,Z 259.897,A -85,B 0,C 180,E1 -12553.533,E2 -12553.533} C_VEL
LIN {X 0,Y 369.002,Z 260.018,A -85,B 0,C 180,E1 -12554.442,E2 -12554.442} C_VEL
LIN {X 0,Y 368.942,Z 260.024,A -85,B 0,C 180,E1 -12554.749,E2 -12554.749} C_VEL
LIN {X 0,Y 368.903,Z 260.032,A -85,B 0,C 180,E1 -12558.192,E2 -12558.192} C_VEL
LIN {X 0,Y 368.872,Z 260.036,A -85,B 0,C 180,E1 -12561.365,E2 -12561.365} C_VEL
LIN {X 0,Y 368.899,Z 260.032,A -85,B 0,C 180,E1 -12565.153,E2 -12565.153} C_VEL
LIN {X 0,Y 368.879,Z 260.034,A -85,B 0,C 180,E1 -12569.051,E2 -12569.051} C_VEL
LIN {X 0,Y 368.931,Z 260.027,A -85,B 0,C 180,E1 -12572.803,E2 -12572.803} C_VEL
LIN {X 0,Y 368.905,Z 260.029,A -85,B 0,C 180,E1 -12576.124,E2 -12576.124} C_VEL
LIN {X 0,Y 368.904,Z 260.03,A -85,B 0,C 180,E1 -12579.953,E2 -12579.953} C_VEL
LIN {X 0,Y 368.946,Z 260.028,A -85,B 0,C 180,E1 -12583.405,E2 -12583.405} C_VEL
LIN {X 0,Y 369.039,Z 260.016,A -85,B 0,C 180,E1 -12586.797,E2 -12586.797} C_VEL
LIN {X 0,Y 369.046,Z 260.012,A -85,B 0,C 180,E1 -12590.138,E2 -12590.138} C_VEL
LIN {X 0,Y 369.165,Z 259.998,A -85,B 0,C 180,E1 -12593.448,E2 -12593.448} C_VEL
LIN {X 0,Y 369.304,Z 259.979,A -85,B 0,C 180,E1 -12597.825,E2 -12597.825} C_VEL
LIN {X 0,Y 369.444,Z 259.962,A -85,B 0,C 180,E1 -12600.006,E2 -12600.006} C_VEL
LIN {X 0,Y 369.295,Z 259.982,A -85,B 0,C 180,E1 -12602.188,E2 -12602.188} C_VEL
LIN {X 0,Y 369.173,Z 260.002,A -85,B 0,C 180,E1 -12606.565,E2 -12606.565} C_VEL
LIN {X 0,Y 369.059,Z 260.011,A -85,B 0,C 180,E1 -12609.874,E2 -12609.874} C_VEL
LIN {X 0,Y 369.037,Z 260.013,A -85,B 0,C 180,E1 -12613.778,E2 -12613.778} C_VEL
LIN {X 0,Y 368.993,Z 260.019,A -85,B 0,C 180,E1 -12617.748,E2 -12617.748} C_VEL
LIN {X 0,Y 368.913,Z 260.028,A -85,B 0,C 180,E1 -12621.226,E2 -12621.226} C_VEL
LIN {X 0,Y 368.926,Z 260.03,A -85,B 0,C 180,E1 -12623.883,E2 -12623.883} C_VEL
LIN {X 0,Y 368.875,Z 260.033,A -85,B 0,C 180,E1 -12627.216,E2 -12627.216} C_VEL
LIN {X 0,Y 368.902,Z 260.032,A -85,B 0,C 180,E1 -12629.697,E2 -12629.697} C_VEL
LIN {X 0,Y 368.905,Z 260.029,A -85,B 0,C 180,E1 -12633.047,E2 -12633.047} C_VEL
LIN {X 0,Y 368.921,Z 260.033,A -85,B 0,C 180,E1 -12636.202,E2 -12636.202} C_VEL
LIN {X 0,Y 368.949,Z 260.307,A -85,B 0,C 180,E1 -12637.563,E2 -12637.563} C_VEL
LIN {X 0,Y 369.278,Z 262.592,A -85,B 0,C 180,E1 -12640.425,E2 -12640.425} C_VEL
LIN {X 0,Y 369.705,Z 265.523,A -85,B 0,C 180,E1 -12643.751,E2 -12643.751} C_VEL
LIN {X 0,Y 369.955,Z 268.48,A -85,B 0,C 180,E1 -12646.853,E2 -12646.853} C_VEL
LIN {X 0,Y 369.796,Z 271.488,A -85,B 0,C 180,E1 -12649.748,E2 -12649.748} C_VEL
LIN {X 0,Y 369.469,Z 275.143,A -85,B 0,C 180,E1 -12653.033,E2 -12653.033} C_VEL
LIN {X 0,Y 369.061,Z 279.206,A -85,B 0,C 180,E1 -12656.48,E2 -12656.48} C_VEL
LIN {X 0,Y 368.739,Z 282.399,A -85,B 0,C 180,E1 -12659.063,E2 -12659.063} C_VEL
LIN {X 0,Y 368.251,Z 287.116,A -85,B 0,C 180,E1 -12662.74,E2 -12662.74} C_VEL
LIN {X 0,Y 367.961,Z 292.094,A -85,B 0,C 180,E1 -12666.47,E2 -12666.47} C_VEL
LIN {X 0,Y 367.669,Z 297.404,A -85,B 0,C 180,E1 -12670.349,E2 -12670.349} C_VEL
LIN {X 0,Y 369.825,Z 307.696,A -85,B 0,C 180,E1 -12670.825,E2 -12670.825} C_VEL
LIN {X 0,Y 371.536,Z 317.057,A -85,B 0,C 180,E1 -12671.368,E2 -12671.368} C_VEL
LIN {X 0,Y 372.861,Z 326.404,A -85,B 0,C 180,E1 -12672.016,E2 -12672.016} C_VEL
LIN {X 0,Y 373.41,Z 332.394,A -85,B 0,C 180,E1 -12672.474,E2 -12672.474} C_VEL
LIN {X 0,Y 372.475,Z 343.305,A -85,B 0,C 180,E1 -12673.419,E2 -12673.419} C_VEL
LIN {X 0,Y 371.578,Z 352.249,A -85,B 0,C 180,E1 -12674.364,E2 -12674.364} C_VEL
LIN {X 0,Y 370.937,Z 359.411,A -85,B 0,C 180,E1 -12675.261,E2 -12675.261} C_VEL
LIN {X 0,Y 370.091,Z 368.002,A -85,B 0,C 180,E1 -12676.549,E2 -12676.549} C_VEL
LIN {X 0,Y 369.436,Z 374.204,A -85,B 0,C 180,E1 -12677.643,E2 -12677.643} C_VEL
LIN {X 0,Y 368.707,Z 380.74,A -85,B 0,C 180,E1 -12679.012,E2 -12679.012} C_VEL
LIN {X 0,Y 368.3,Z 385.242,A -85,B 0,C 180,E1 -12680.111,E2 -12680.111} C_VEL
LIN {X 0,Y 367.858,Z 390.735,A -85,B 0,C 180,E1 -12681.762,E2 -12681.762} C_VEL
LIN {X 0,Y 367.58,Z 395.06,A -85,B 0,C 180,E1 -12683.413,E2 -12683.413} C_VEL
LIN {X 0,Y 367.476,Z 397.427,A -85,B 0,C 180,E1 -12684.513,E2 -12684.513} C_VEL
LIN {X 0,Y 367.439,Z 399.226,A -85,B 0,C 180,E1 -12685.612,E2 -12685.612} C_VEL
LIN {X 0,Y 367.363,Z 401.67,A -85,B 0,C 180,E1 -12687.807,E2 -12687.807} C_VEL
LIN {X 0,Y 367.399,Z 402.26,A -85,B 0,C 180,E1 -12688.904,E2 -12688.904} C_VEL
LIN {X 0,Y 367.399,Z 402.26,A -85,B 0,C 180,E1 -12691.096,E2 -12691.096} C_VEL
LIN {X 0,Y 367.363,Z 401.67,A -85,B 0,C 180,E1 -12692.193,E2 -12692.193} C_VEL
LIN {X 0,Y 367.439,Z 399.226,A -85,B 0,C 180,E1 -12694.388,E2 -12694.388} C_VEL
LIN {X 0,Y 367.492,Z 396.344,A -85,B 0,C 180,E1 -12696.007,E2 -12696.007} C_VEL
LIN {X 0,Y 367.735,Z 392.288,A -85,B 0,C 180,E1 -12697.688,E2 -12697.688} C_VEL
LIN {X 0,Y 368.122,Z 387.158,A -85,B 0,C 180,E1 -12699.339,E2 -12699.339} C_VEL
LIN {X 0,Y 368.616,Z 381.896,A -85,B 0,C 180,E1 -12700.713,E2 -12700.713} C_VEL
LIN {X 0,Y 369.261,Z 375.579,A -85,B 0,C 180,E1 -12702.084,E2 -12702.084} C_VEL
LIN {X 0,Y 369.929,Z 369.629,A -85,B 0,C 180,E1 -12703.178,E2 -12703.178} C_VEL
LIN {X 0,Y 370.588,Z 362.701,A -85,B 0,C 180,E1 -12704.272,E2 -12704.272} C_VEL
LIN {X 0,Y 371.341,Z 354.518,A -85,B 0,C 180,E1 -12705.364,E2 -12705.364} C_VEL
LIN {X 0,Y 372.19,Z 346.007,A -85,B 0,C 180,E1 -12706.312,E2 -12706.312} C_VEL
LIN {X 0,Y 373.001,Z 337.292,A -85,B 0,C 180,E1 -12707.121,E2 -12707.121} C_VEL
LIN {X 0,Y 373.399,Z 331.318,A -85,B 0,C 180,E1 -12707.612,E2 -12707.612} C_VEL
LIN {X 0,Y 371.905,Z 319.33,A -85,B 0,C 180,E1 -12708.487,E2 -12708.487} C_VEL
LIN {X 0,Y 370.032,Z 308.731,A -85,B 0,C 180,E1 -12709.122,E2 -12709.122} C_VEL
LIN {X 0,Y 367.825,Z 298.593,A -85,B 0,C 180,E1 -12709.611,E2 -12709.611} C_VEL
LIN {X 0,Y 367.667,Z 297.344,A -85,B 0,C 180,E1 -12709.684,E2 -12709.684} C_VEL
LIN {X 0,Y 367.964,Z 291.927,A -85,B 0,C 180,E1 -12713.646,E2 -12713.646} C_VEL
LIN {X 0,Y 368.251,Z 287.107,A -85,B 0,C 180,E1 -12717.26,E2 -12717.26} C_VEL
LIN {X 0,Y 368.745,Z 282.343,A -85,B 0,C 180,E1 -12720.97,E2 -12720.97} C_VEL
LIN {X 0,Y 369.064,Z 279.204,A -85,B 0,C 180,E1 -12723.52,E2 -12723.52} C_VEL
LIN {X 0,Y 369.467,Z 275.137,A -85,B 0,C 180,E1 -12726.967,E2 -12726.967} C_VEL
LIN {X 0,Y 369.822,Z 271.201,A -85,B 0,C 180,E1 -12730.517,E2 -12730.517} C_VEL
LIN {X 0,Y 369.967,Z 268.466,A -85,B 0,C 180,E1 -12733.145,E2 -12733.145} C_VEL
LIN {X 0,Y 369.701,Z 265.523,A -85,B 0,C 180,E1 -12736.25,E2 -12736.25} C_VEL
LIN {X 0,Y 369.265,Z 262.512,A -85,B 0,C 180,E1 -12739.671,E2 -12739.671} C_VEL
LIN {X 0,Y 368.95,Z 260.308,A -85,B 0,C 180,E1 -12742.437,E2 -12742.437} C_VEL
LIN {X 0,Y 368.936,Z 260.032,A -85,B 0,C 180,E1 -12744.995,E2 -12744.995} C_VEL
LIN {X 0,Y 368.905,Z 260.033,A -85,B 0,C 180,E1 -12747.757,E2 -12747.757} C_VEL
LIN {X 0,Y 368.92,Z 260.03,A -85,B 0,C 180,E1 -12751.554,E2 -12751.554} C_VEL
LIN {X 0,Y 368.905,Z 260.03,A -85,B 0,C 180,E1 -12755.216,E2 -12755.216} C_VEL
LIN {X 0,Y 368.925,Z 260.031,A -85,B 0,C 180,E1 -12757.599,E2 -12757.599} C_VEL
LIN {X 0,Y 368.956,Z 260.024,A -85,B 0,C 180,E1 -12761.1,E2 -12761.1} C_VEL
LIN {X 0,Y 368.997,Z 260.018,A -85,B 0,C 180,E1 -12764.53,E2 -12764.53} C_VEL
LIN {X 0,Y 369.002,Z 260.02,A -85,B 0,C 180,E1 -12767.901,E2 -12767.901} C_VEL
LIN {X 0,Y 369.142,Z 260.002,A -85,B 0,C 180,E1 -12771.886,E2 -12771.886} C_VEL
LIN {X 0,Y 369.122,Z 260.002,A -85,B 0,C 180,E1 -12774.531,E2 -12774.531} C_VEL
LIN {X 0,Y 369.295,Z 259.982,A -85,B 0,C 180,E1 -12777.812,E2 -12777.812} C_VEL
LIN {X 0,Y 369.444,Z 259.962,A -85,B 0,C 180,E1 -12779.994,E2 -12779.994} C_VEL
LIN {X 0,Y 369.304,Z 259.979,A -85,B 0,C 180,E1 -12782.175,E2 -12782.175} C_VEL
LIN {X 0,Y 369.164,Z 259.998,A -85,B 0,C 180,E1 -12786.56,E2 -12786.56} C_VEL
LIN {X 0,Y 369.046,Z 260.012,A -85,B 0,C 180,E1 -12789.862,E2 -12789.862} C_VEL
LIN {X 0,Y 369.018,Z 260.015,A -85,B 0,C 180,E1 -12793.765,E2 -12793.765} C_VEL
LIN {X 0,Y 368.968,Z 260.021,A -85,B 0,C 180,E1 -12797.736,E2 -12797.736} C_VEL
LIN {X 0,Y 368.884,Z 260.033,A -85,B 0,C 180,E1 -12801.214,E2 -12801.214} C_VEL
LIN {X 0,Y 368.925,Z 260.031,A -85,B 0,C 180,E1 -12804.769,E2 -12804.769} C_VEL
LIN {X 0,Y 368.931,Z 260.027,A -85,B 0,C 180,E1 -12807.197,E2 -12807.197} C_VEL
LIN {X 0,Y 368.877,Z 260.034,A -85,B 0,C 180,E1 -12810.981,E2 -12810.981} C_VEL
LIN {X 0,Y 368.899,Z 260.032,A -85,B 0,C 180,E1 -12814.847,E2 -12814.847} C_VEL
LIN {X 0,Y 368.872,Z 260.036,A -85,B 0,C 180,E1 -12818.635,E2 -12818.635} C_VEL
LIN {X 0,Y 368.909,Z 260.033,A -85,B 0,C 180,E1 -12822.016,E2 -12822.016} C_VEL
LIN {X 0,Y 368.947,Z 260.024,A -85,B 0,C 180,E1 -12825.188,E2 -12825.188} C_VEL
LIN {X 0,Y 368.894,Z 260.035,A -85,B 0,C 180,E1 -12828.18,E2 -12828.18} C_VEL
LIN {X 0,Y 368.863,Z 260.035,A -85,B 0,C 180,E1 -12831.354,E2 -12831.354} C_VEL
LIN {X 0,Y 368.884,Z 260.032,A -85,B 0,C 180,E1 -12835.142,E2 -12835.142} C_VEL
LIN {X 0,Y 368.875,Z 260.033,A -85,B 0,C 180,E1 -12839.042,E2 -12839.042} C_VEL
LIN {X 0,Y 368.93,Z 260.031,A -85,B 0,C 180,E1 -12841.561,E2 -12841.561} C_VEL
LIN {X 0,Y 368.904,Z 260.032,A -85,B 0,C 180,E1 -12845.221,E2 -12845.221} C_VEL
LIN {X 0,Y 368.932,Z 260.027,A -85,B 0,C 180,E1 -12848.949,E2 -12848.949} C_VEL
LIN {X 0,Y 368.932,Z 260.03,A -85,B 0,C 180,E1 -12852.255,E2 -12852.255} C_VEL
LIN {X 0,Y 368.983,Z 260.208,A -85,B 0,C 180,E1 -12855.418,E2 -12855.418} C_VEL
LIN {X 0,Y 369.9,Z 262.79,A -85,B 0,C 180,E1 -12855.734,E2 -12855.734} C_VEL
LIN {X 0,Y 371.765,Z 264.825,A -85,B 0,C 180,E1 -12856.311,E2 -12856.311} C_VEL
LIN {X 0,Y 373.66,Z 266.063,A -85,B 0,C 180,E1 -12856.886,E2 -12856.886} C_VEL
LIN {X 0,Y 375.396,Z 268.944,A -85,B 0,C 180,E1 -12857.498,E2 -12857.498} C_VEL
LIN {X 0,Y 378.003,Z 271.257,A -85,B 0,C 180,E1 -12858.416,E2 -12858.416} C_VEL
LIN {X 0,Y 379.317,Z 272.104,A -85,B 0,C 180,E1 -12858.887,E2 -12858.887} C_VEL
LIN {X 0,Y 381.078,Z 274.813,A -85,B 0,C 180,E1 -12859.641,E2 -12859.641} C_VEL
LIN {X 0,Y 383.643,Z 277.056,A -85,B 0,C 180,E1 -12860.754,E2 -12860.754} C_VEL
LIN {X 0,Y 386.028,Z 278.396,A -85,B 0,C 180,E1 -12861.879,E2 -12861.879} C_VEL
LIN {X 0,Y 387.954,Z 281.231,A -85,B 0,C 180,E1 -12863.046,E2 -12863.046} C_VEL
LIN {X 0,Y 389.984,Z 283.187,A -85,B 0,C 180,E1 -12864.442,E2 -12864.442} C_VEL
LIN {X 0,Y 391.64,Z 284.168,A -85,B 0,C 180,E1 -12865.884,E2 -12865.884} C_VEL
LIN {X 0,Y 393.217,Z 284.545,A -85,B 0,C 180,E1 -12867.952,E2 -12867.952} C_VEL
LIN {X 0,Y 393.777,Z 284.603,A -85,B 0,C 180,E1 -12870,E2 -12870} C_VEL
LIN {X 0,Y 393.217,Z 284.545,A -85,B 0,C 180,E1 -12872.048,E2 -12872.048} C_VEL
LIN {X 0,Y 391.64,Z 284.169,A -85,B 0,C 180,E1 -12874.116,E2 -12874.116} C_VEL
LIN {X 0,Y 389.612,Z 282.895,A -85,B 0,C 180,E1 -12875.823,E2 -12875.823} C_VEL
LIN {X 0,Y 387.556,Z 280.705,A -85,B 0,C 180,E1 -12877.216,E2 -12877.216} C_VEL
LIN {X 0,Y 385.892,Z 278.104,A -85,B 0,C 180,E1 -12878.208,E2 -12878.208} C_VEL
LIN {X 0,Y 383.075,Z 276.63,A -85,B 0,C 180,E1 -12879.504,E2 -12879.504} C_VEL
LIN {X 0,Y 380.644,Z 274.274,A -85,B 0,C 180,E1 -12880.539,E2 -12880.539} C_VEL
LIN {X 0,Y 379.096,Z 271.754,A -85,B 0,C 180,E1 -12881.204,E2 -12881.204} C_VEL
LIN {X 0,Y 376.44,Z 270.076,A -85,B 0,C 180,E1 -12882.124,E2 -12882.124} C_VEL
LIN {X 0,Y 374.361,Z 267.451,A -85,B 0,C 180,E1 -12882.868,E2 -12882.868} C_VEL
LIN {X 0,Y 373.42,Z 265.746,A -85,B 0,C 180,E1 -12883.192,E2 -12883.192} C_VEL
LIN {X 0,Y 370.867,Z 264.021,A -85,B 0,C 180,E1 -12883.969,E2 -12883.969} C_VEL
LIN {X 0,Y 369.457,Z 261.93,A -85,B 0,C 180,E1 -12884.405,E2 -12884.405} C_VEL
LIN {X 0,Y 368.961,Z 260.029,A -85,B 0,C 180,E1 -12884.618,E2 -12884.618} C_VEL
LIN {X 0,Y 368.941,Z 260.029,A -85,B 0,C 180,E1 -12887.771,E2 -12887.771} C_VEL
LIN {X 0,Y 368.928,Z 260.027,A -85,B 0,C 180,E1 -12891.219,E2 -12891.219} C_VEL
LIN {X 0,Y 368.904,Z 260.032,A -85,B 0,C 180,E1 -12894.779,E2 -12894.779} C_VEL
LIN {X 0,Y 368.93,Z 260.031,A -85,B 0,C 180,E1 -12898.439,E2 -12898.439} C_VEL
LIN {X 0,Y 368.844,Z 260.043,A -85,B 0,C 180,E1 -12902.242,E2 -12902.242} C_VEL
LIN {X 0,Y 368.876,Z 260.033,A -85,B 0,C 180,E1 -12905.006,E2 -12905.006} C_VEL
LIN {X 0,Y 368.863,Z 260.035,A -85,B 0,C 180,E1 -12908.646,E2 -12908.646} C_VEL
LIN {X 0,Y 368.895,Z 260.036,A -85,B 0,C 180,E1 -12912.025,E2 -12912.025} C_VEL
LIN {X 0,Y 368.942,Z 260.024,A -85,B 0,C 180,E1 -12914.749,E2 -12914.749} C_VEL
LIN {X 0,Y 368.325,Z 260.106,A -85,B 0,C 180,E1 -12915.66,E2 -12915.66} C_VEL
LIN {X 0,Y 365.472,Z 260.461,A -85,B 0,C 180,E1 -12917.14,E2 -12917.14} C_VEL
LIN {X 0,Y 363.012,Z 260.765,A -85,B 0,C 180,E1 -12918.337,E2 -12918.337} C_VEL
LIN {X 0,Y 361.939,Z 260.898,A -85,B 0,C 180,E1 -12919.264,E2 -12919.264} C_VEL
LIN {X 0,Y 361.845,Z 260.909,A -85,B 0,C 180,E1 -12919.578,E2 -12919.578} C_VEL
LIN {X 0,Y 361.83,Z 260.911,A -85,B 0,C 180,E1 -12922.988,E2 -12922.988} C_VEL
LIN {X 0,Y 361.825,Z 260.911,A -85,B 0,C 180,E1 -12926.637,E2 -12926.637} C_VEL
LIN {X 0,Y 361.826,Z 260.915,A -85,B 0,C 180,E1 -12929.677,E2 -12929.677} C_VEL
LIN {X 0,Y 361.923,Z 260.905,A -85,B 0,C 180,E1 -12933.482,E2 -12933.482} C_VEL
LIN {X 0,Y 361.852,Z 260.912,A -85,B 0,C 180,E1 -12937.151,E2 -12937.151} C_VEL
LIN {X 0,Y 361.859,Z 260.908,A -85,B 0,C 180,E1 -12940.729,E2 -12940.729} C_VEL
LIN {X 0,Y 361.921,Z 260.899,A -85,B 0,C 180,E1 -12944.233,E2 -12944.233} C_VEL
LIN {X 0,Y 361.98,Z 260.893,A -85,B 0,C 180,E1 -12946.535,E2 -12946.535} C_VEL
LIN {X 0,Y 361.983,Z 260.891,A -85,B 0,C 180,E1 -12949.944,E2 -12949.944} C_VEL
LIN {X 0,Y 362.127,Z 260.876,A -85,B 0,C 180,E1 -12953.32,E2 -12953.32} C_VEL
LIN {X 0,Y 362.268,Z 260.856,A -85,B 0,C 180,E1 -12957.783,E2 -12957.783} C_VEL
LIN {X 0,Y 362.393,Z 260.841,A -85,B 0,C 180,E1 -12960.006,E2 -12960.006} C_VEL
LIN {X 0,Y 362.259,Z 260.859,A -85,B 0,C 180,E1 -12962.23,E2 -12962.23} C_VEL
LIN {X 0,Y 362.136,Z 260.878,A -85,B 0,C 180,E1 -12966.693,E2 -12966.693} C_VEL
LIN {X 0,Y 361.996,Z 260.892,A -85,B 0,C 180,E1 -12970.069,E2 -12970.069} C_VEL
LIN {X 0,Y 361.998,Z 260.891,A -85,B 0,C 180,E1 -12973.904,E2 -12973.904} C_VEL
LIN {X 0,Y 361.93,Z 260.899,A -85,B 0,C 180,E1 -12976.94,E2 -12976.94} C_VEL
LIN {X 0,Y 361.887,Z 260.907,A -85,B 0,C 180,E1 -12980.467,E2 -12980.467} C_VEL
LIN {X 0,Y 361.883,Z 260.91,A -85,B 0,C 180,E1 -12984.112,E2 -12984.112} C_VEL
LIN {X 0,Y 361.849,Z 260.911,A -85,B 0,C 180,E1 -12987.789,E2 -12987.789} C_VEL
LIN {X 0,Y 361.855,Z 260.908,A -85,B 0,C 180,E1 -12991.29,E2 -12991.29} C_VEL
LIN {X 0,Y 361.86,Z 260.914,A -85,B 0,C 180,E1 -12994.285,E2 -12994.285} C_VEL
LIN {X 0,Y 361.91,Z 261.193,A -85,B 0,C 180,E1 -12997.234,E2 -12997.234} C_VEL
LIN {X 0,Y 362.38,Z 264.419,A -85,B 0,C 180,E1 -13001.259,E2 -13001.259} C_VEL
LIN {X 0,Y 362.724,Z 266.994,A -85,B 0,C 180,E1 -13004.234,E2 -13004.234} C_VEL
LIN {X 0,Y 362.888,Z 268.451,A -85,B 0,C 180,E1 -13005.798,E2 -13005.798} C_VEL
LIN {X 0,Y 362.837,Z 271.446,A -85,B 0,C 180,E1 -13008.811,E2 -13008.811} C_VEL
LIN {X 0,Y 362.553,Z 274.49,A -85,B 0,C 180,E1 -13011.662,E2 -13011.662} C_VEL
LIN {X 0,Y 362.234,Z 277.771,A -85,B 0,C 180,E1 -13014.581,E2 -13014.581} C_VEL
LIN {X 0,Y 361.922,Z 280.687,A -85,B 0,C 180,E1 -13017.064,E2 -13017.064} C_VEL
LIN {X 0,Y 361.557,Z 283.829,A -85,B 0,C 180,E1 -13019.643,E2 -13019.643} C_VEL
LIN {X 0,Y 361.103,Z 288.783,A -85,B 0,C 180,E1 -13023.552,E2 -13023.552} C_VEL
LIN {X 0,Y 360.793,Z 293.39,A -85,B 0,C 180,E1 -13027.072,E2 -13027.072} C_VEL
LIN {X 0,Y 360.605,Z 297.204,A -85,B 0,C 180,E1 -13029.933,E2 -13029.933} C_VEL
LIN {X 0,Y 363.451,Z 310.717,A -85,B 0,C 180,E1 -13030.609,E2 -13030.609} C_VEL
LIN {X 0,Y 365.629,Z 324.105,A -85,B 0,C 180,E1 -13031.498,E2 -13031.498} C_VEL
LIN {X 0,Y 366.514,Z 332.195,A -85,B 0,C 180,E1 -13032.134,E2 -13032.134} C_VEL
LIN {X 0,Y 365.68,Z 343.11,A -85,B 0,C 180,E1 -13033.101,E2 -13033.101} C_VEL
LIN {X 0,Y 364.715,Z 352.053,A -85,B 0,C 180,E1 -13034.063,E2 -13034.063} C_VEL
LIN {X 0,Y 363.973,Z 359.945,A -85,B 0,C 180,E1 -13035.081,E2 -13035.081} C_VEL
LIN {X 0,Y 363.154,Z 367.806,A -85,B 0,C 180,E1 -13036.287,E2 -13036.287} C_VEL
LIN {X 0,Y 362.468,Z 374.008,A -85,B 0,C 180,E1 -13037.401,E2 -13037.401} C_VEL
LIN {X 0,Y 361.695,Z 380.544,A -85,B 0,C 180,E1 -13038.796,E2 -13038.796} C_VEL
LIN {X 0,Y 361.275,Z 385.047,A -85,B 0,C 180,E1 -13039.917,E2 -13039.917} C_VEL
LIN {X 0,Y 360.807,Z 390.539,A -85,B 0,C 180,E1 -13041.6,E2 -13041.6} C_VEL
LIN {X 0,Y 360.515,Z 394.865,A -85,B 0,C 180,E1 -13043.283,E2 -13043.283} C_VEL
LIN {X 0,Y 360.401,Z 397.232,A -85,B 0,C 180,E1 -13044.405,E2 -13044.405} C_VEL
LIN {X 0,Y 360.352,Z 399.031,A -85,B 0,C 180,E1 -13045.526,E2 -13045.526} C_VEL
LIN {X 0,Y 360.268,Z 401.476,A -85,B 0,C 180,E1 -13047.764,E2 -13047.764} C_VEL
LIN {X 0,Y 360.299,Z 402.065,A -85,B 0,C 180,E1 -13048.882,E2 -13048.882} C_VEL
LIN {X 0,Y 360.299,Z 402.065,A -85,B 0,C 180,E1 -13051.118,E2 -13051.118} C_VEL
LIN {X 0,Y 360.268,Z 401.476,A -85,B 0,C 180,E1 -13052.236,E2 -13052.236} C_VEL
LIN {X 0,Y 360.351,Z 399.031,A -85,B 0,C 180,E1 -13054.474,E2 -13054.474} C_VEL
LIN {X 0,Y 360.395,Z 396.506,A -85,B 0,C 180,E1 -13055.961,E2 -13055.961} C_VEL
LIN {X 0,Y 360.607,Z 393.625,A -85,B 0,C 180,E1 -13057.278,E2 -13057.278} C_VEL
LIN {X 0,Y 360.934,Z 388.879,A -85,B 0,C 180,E1 -13058.961,E2 -13058.961} C_VEL
LIN {X 0,Y 361.515,Z 382.857,A -85,B 0,C 180,E1 -13060.642,E2 -13060.642} C_VEL
LIN {X 0,Y 362.114,Z 376.759,A -85,B 0,C 180,E1 -13062.042,E2 -13062.042} C_VEL
LIN {X 0,Y 362.808,Z 371.061,A -85,B 0,C 180,E1 -13063.156,E2 -13063.156} C_VEL
LIN {X 0,Y 363.695,Z 362.505,A -85,B 0,C 180,E1 -13064.549,E2 -13064.549} C_VEL
LIN {X 0,Y 364.467,Z 354.323,A -85,B 0,C 180,E1 -13065.662,E2 -13065.662} C_VEL
LIN {X 0,Y 365.381,Z 345.813,A -85,B 0,C 180,E1 -13066.625,E2 -13066.625} C_VEL
LIN {X 0,Y 366.217,Z 337.097,A -85,B 0,C 180,E1 -13067.449,E2 -13067.449} C_VEL
LIN {X 0,Y 366.45,Z 331.206,A -85,B 0,C 180,E1 -13067.95,E2 -13067.95} C_VEL
LIN {X 0,Y 364.983,Z 319.65,A -85,B 0,C 180,E1 -13068.822,E2 -13068.822} C_VEL
LIN {X 0,Y 362.988,Z 308.296,A -85,B 0,C 180,E1 -13069.518,E2 -13069.518} C_VEL
LIN {X 0,Y 360.597,Z 297.174,A -85,B 0,C 180,E1 -13070.09,E2 -13070.09} C_VEL
LIN {X 0,Y 360.908,Z 291.777,A -85,B 0,C 180,E1 -13074.137,E2 -13074.137} C_VEL
LIN {X 0,Y 361.22,Z 286.987,A -85,B 0,C 180,E1 -13077.836,E2 -13077.836} C_VEL
LIN {X 0,Y 361.734,Z 282.248,A -85,B 0,C 180,E1 -13081.639,E2 -13081.639} C_VEL
LIN {X 0,Y 362.086,Z 279.122,A -85,B 0,C 180,E1 -13084.254,E2 -13084.254} C_VEL
LIN {X 0,Y 362.474,Z 275.578,A -85,B 0,C 180,E1 -13087.344,E2 -13087.344} C_VEL
LIN {X 0,Y 362.838,Z 271.442,A -85,B 0,C 180,E1 -13091.189,E2 -13091.189} C_VEL
LIN {X 0,Y 362.886,Z 268.412,A -85,B 0,C 180,E1 -13094.222,E2 -13094.222} C_VEL
LIN {X 0,Y 362.503,Z 265.535,A -85,B 0,C 180,E1 -13097.451,E2 -13097.451} C_VEL
LIN {X 0,Y 362.084,Z 262.609,A -85,B 0,C 180,E1 -13100.93,E2 -13100.93} C_VEL
LIN {X 0,Y 361.885,Z 261.038,A -85,B 0,C 180,E1 -13102.979,E2 -13102.979} C_VEL
LIN {X 0,Y 361.867,Z 260.907,A -85,B 0,C 180,E1 -13106.627,E2 -13106.627} C_VEL
LIN {X 0,Y 361.864,Z 260.909,A -85,B 0,C 180,E1 -13109.666,E2 -13109.666} C_VEL
LIN {X 0,Y 361.87,Z 260.908,A -85,B 0,C 180,E1 -13113.463,E2 -13113.463} C_VEL
LIN {X 0,Y 361.881,Z 260.905,A -85,B 0,C 180,E1 -13117.139,E2 -13117.139} C_VEL
LIN {X 0,Y 361.886,Z 260.903,A -85,B 0,C 180,E1 -13120.717,E2 -13120.717} C_VEL
LIN {X 0,Y 361.944,Z 260.897,A -85,B 0,C 180,E1 -13124.22,E2 -13124.22} C_VEL
LIN {X 0,Y 361.999,Z 260.889,A -85,B 0,C 180,E1 -13126.522,E2 -13126.522} C_VEL
LIN {X 0,Y 361.996,Z 260.892,A -85,B 0,C 180,E1 -13129.931,E2 -13129.931} C_VEL
LIN {X 0,Y 362.136,Z 260.878,A -85,B 0,C 180,E1 -13133.307,E2 -13133.307} C_VEL
LIN {X 0,Y 362.259,Z 260.859,A -85,B 0,C 180,E1 -13137.77,E2 -13137.77} C_VEL
LIN {X 0,Y 362.393,Z 260.841,A -85,B 0,C 180,E1 -13139.994,E2 -13139.994} C_VEL
LIN {X 0,Y 362.268,Z 260.856,A -85,B 0,C 180,E1 -13142.217,E2 -13142.217} C_VEL
LIN {X 0,Y 362.127,Z 260.876,A -85,B 0,C 180,E1 -13146.68,E2 -13146.68} C_VEL
LIN {X 0,Y 361.983,Z 260.891,A -85,B 0,C 180,E1 -13150.056,E2 -13150.056} C_VEL
LIN {X 0,Y 361.979,Z 260.892,A -85,B 0,C 180,E1 -13153.892,E2 -13153.892} C_VEL
LIN {X 0,Y 361.906,Z 260.906,A -85,B 0,C 180,E1 -13156.927,E2 -13156.927} C_VEL
LIN {X 0,Y 361.858,Z 260.91,A -85,B 0,C 180,E1 -13160.454,E2 -13160.454} C_VEL
LIN {X 0,Y 361.866,Z 260.907,A -85,B 0,C 180,E1 -13164.106,E2 -13164.106} C_VEL
LIN {X 0,Y 361.911,Z 260.905,A -85,B 0,C 180,E1 -13166.714,E2 -13166.714} C_VEL
LIN {X 0,Y 361.826,Z 260.915,A -85,B 0,C 180,E1 -13170.323,E2 -13170.323} C_VEL
LIN {X 0,Y 361.818,Z 260.917,A -85,B 0,C 180,E1 -13174.274,E2 -13174.274} C_VEL
LIN {X 0,Y 361.826,Z 260.911,A -85,B 0,C 180,E1 -13177.217,E2 -13177.217} C_VEL
LIN {X 0,Y 361.865,Z 260.907,A -85,B 0,C 180,E1 -13180.762,E2 -13180.762} C_VEL
LIN {X 0,Y 361.89,Z 260.907,A -85,B 0,C 180,E1 -13184.345,E2 -13184.345} C_VEL
LIN {X 0,Y 361.84,Z 260.911,A -85,B 0,C 180,E1 -13187.554,E2 -13187.554} C_VEL
LIN {X 0,Y 361.825,Z 260.911,A -85,B 0,C 180,E1 -13190.967,E2 -13190.967} C_VEL
LIN {X 0,Y 361.822,Z 260.912,A -85,B 0,C 180,E1 -13194.651,E2 -13194.651} C_VEL
LIN {X 0,Y 361.784,Z 260.917,A -85,B 0,C 180,E1 -13198.366,E2 -13198.366} C_VEL
LIN {X 0,Y 361.846,Z 260.909,A -85,B 0,C 180,E1 -13200.951,E2 -13200.951} C_VEL
LIN {X 0,Y 361.898,Z 260.906,A -85,B 0,C 180,E1 -13203.471,E2 -13203.471} C_VEL
LIN {X 0,Y 361.864,Z 260.908,A -85,B 0,C 180,E1 -13207.144,E2 -13207.144} C_VEL
LIN {X 0,Y 361.875,Z 260.907,A -85,B 0,C 180,E1 -13210.722,E2 -13210.722} C_VEL
LIN {X 0,Y 361.89,Z 260.967,A -85,B 0,C 180,E1 -13213.772,E2 -13213.772} C_VEL
LIN {X 0,Y 362.756,Z 263.566,A -85,B 0,C 180,E1 -13214.054,E2 -13214.054} C_VEL
LIN {X 0,Y 364.722,Z 265.74,A -85,B 0,C 180,E1 -13214.572,E2 -13214.572} C_VEL
LIN {X 0,Y 366.195,Z 266.695,A -85,B 0,C 180,E1 -13214.955,E2 -13214.955} C_VEL
LIN {X 0,Y 367.885,Z 269.589,A -85,B 0,C 180,E1 -13215.479,E2 -13215.479} C_VEL
LIN {X 0,Y 370.428,Z 271.832,A -85,B 0,C 180,E1 -13216.21,E2 -13216.21} C_VEL
LIN {X 0,Y 371.519,Z 272.788,A -85,B 0,C 180,E1 -13216.552,E2 -13216.552} C_VEL
LIN {X 0,Y 373.892,Z 275.989,A -85,B 0,C 180,E1 -13217.343,E2 -13217.343} C_VEL
LIN {X 0,Y 376.758,Z 278.232,A -85,B 0,C 180,E1 -13218.322,E2 -13218.322} C_VEL
LIN {X 0,Y 377.605,Z 278.983,A -85,B 0,C 180,E1 -13218.62,E2 -13218.62} C_VEL
LIN {X 0,Y 380.036,Z 282.092,A -85,B 0,C 180,E1 -13219.613,E2 -13219.613} C_VEL
LIN {X 0,Y 382.942,Z 284.287,A -85,B 0,C 180,E1 -13220.851,E2 -13220.851} C_VEL
LIN {X 0,Y 384.645,Z 285.231,A -85,B 0,C 180,E1 -13221.638,E2 -13221.638} C_VEL
LIN {X 0,Y 386.759,Z 288.132,A -85,B 0,C 180,E1 -13222.868,E2 -13222.868} C_VEL
LIN {X 0,Y 388.889,Z 290.132,A -85,B 0,C 180,E1 -13224.296,E2 -13224.296} C_VEL
LIN {X 0,Y 390.753,Z 291.192,A -85,B 0,C 180,E1 -13225.875,E2 -13225.875} C_VEL
LIN {X 0,Y 392.355,Z 291.591,A -85,B 0,C 180,E1 -13227.947,E2 -13227.947} C_VEL
LIN {X 0,Y 392.772,Z 291.63,A -85,B 0,C 180,E1 -13228.975,E2 -13228.975} C_VEL
LIN {X 0,Y 392.911,Z 291.649,A -85,B 0,C 180,E1 -13230,E2 -13230} C_VEL
LIN {X 0,Y 392.772,Z 291.633,A -85,B 0,C 180,E1 -13231.025,E2 -13231.025} C_VEL
LIN {X 0,Y 391.687,Z 291.421,A -85,B 0,C 180,E1 -13233.086,E2 -13233.086} C_VEL
LIN {X 0,Y 389.885,Z 290.782,A -85,B 0,C 180,E1 -13234.912,E2 -13234.912} C_VEL
LIN {X 0,Y 387.665,Z 289.109,A -85,B 0,C 180,E1 -13236.555,E2 -13236.555} C_VEL
LIN {X 0,Y 385.323,Z 286.34,A -85,B 0,C 180,E1 -13237.967,E2 -13237.967} C_VEL
LIN {X 0,Y 384.27,Z 284.89,A -85,B 0,C 180,E1 -13238.546,E2 -13238.546} C_VEL
LIN {X 0,Y 381.335,Z 283.216,A -85,B 0,C 180,E1 -13239.857,E2 -13239.857} C_VEL
LIN {X 0,Y 378.506,Z 280.329,A -85,B 0,C 180,E1 -13241.012,E2 -13241.012} C_VEL
LIN {X 0,Y 377.298,Z 278.493,A -85,B 0,C 180,E1 -13241.498,E2 -13241.498} C_VEL
LIN {X 0,Y 374.296,Z 276.38,A -85,B 0,C 180,E1 -13242.522,E2 -13242.522} C_VEL
LIN {X 0,Y 371.745,Z 273.186,A -85,B 0,C 180,E1 -13243.369,E2 -13243.369} C_VEL
LIN {X 0,Y 371.003,Z 272.178,A -85,B 0,C 180,E1 -13243.616,E2 -13243.616} C_VEL
LIN {X 0,Y 368.3,Z 270.065,A -85,B 0,C 180,E1 -13244.402,E2 -13244.402} C_VEL
LIN {X 0,Y 366.369,Z 267.109,A -85,B 0,C 180,E1 -13244.987,E2 -13244.987} C_VEL
LIN {X 0,Y 365.807,Z 266.4,A -85,B 0,C 180,E1 -13245.153,E2 -13245.153} C_VEL
LIN {X 0,Y 363.428,Z 264.519,A -85,B 0,C 180,E1 -13245.762,E2 -13245.762} C_VEL
LIN {X 0,Y 362.164,Z 262.188,A -85,B 0,C 180,E1 -13246.125,E2 -13246.125} C_VEL
LIN {X 0,Y 361.878,Z 260.909,A -85,B 0,C 180,E1 -13246.247,E2 -13246.247} C_VEL
LIN {X 0,Y 361.875,Z 260.908,A -85,B 0,C 180,E1 -13249.278,E2 -13249.278} C_VEL
LIN {X 0,Y 361.864,Z 260.908,A -85,B 0,C 180,E1 -13252.856,E2 -13252.856} C_VEL
LIN {X 0,Y 361.886,Z 260.906,A -85,B 0,C 180,E1 -13256.725,E2 -13256.725} C_VEL
LIN {X 0,Y 361.821,Z 260.917,A -85,B 0,C 180,E1 -13260.332,E2 -13260.332} C_VEL
LIN {X 0,Y 361.801,Z 260.919,A -85,B 0,C 180,E1 -13264.285,E2 -13264.285} C_VEL
LIN {X 0,Y 361.815,Z 260.913,A -85,B 0,C 180,E1 -13267.228,E2 -13267.228} C_VEL
LIN {X 0,Y 361.858,Z 260.907,A -85,B 0,C 180,E1 -13270.773,E2 -13270.773} C_VEL
LIN {X 0,Y 361.869,Z 260.906,A -85,B 0,C 180,E1 -13274.744,E2 -13274.744} C_VEL
LIN {X 0,Y 361.849,Z 260.912,A -85,B 0,C 180,E1 -13277.564,E2 -13277.564} C_VEL
LIN {X 0,Y 361.845,Z 260.909,A -85,B 0,C 180,E1 -13279.578,E2 -13279.578} C_VEL
LIN {X 0,Y 361.161,Z 260.995,A -85,B 0,C 180,E1 -13280.506,E2 -13280.506} C_VEL
LIN {X 0,Y 358.312,Z 261.352,A -85,B 0,C 180,E1 -13282.017,E2 -13282.017} C_VEL
LIN {X 0,Y 355.905,Z 261.651,A -85,B 0,C 180,E1 -13283.238,E2 -13283.238} C_VEL
LIN {X 0,Y 354.866,Z 261.78,A -85,B 0,C 180,E1 -13284.183,E2 -13284.183} C_VEL
LIN {X 0,Y 354.777,Z 261.789,A -85,B 0,C 180,E1 -13284.503,E2 -13284.503} C_VEL
LIN {X 0,Y 354.754,Z 261.797,A -85,B 0,C 180,E1 -13287.673,E2 -13287.673} C_VEL
LIN {X 0,Y 354.798,Z 261.791,A -85,B 0,C 180,E1 -13291.624,E2 -13291.624} C_VEL
LIN {X 0,Y 354.869,Z 261.778,A -85,B 0,C 180,E1 -13294.179,E2 -13294.179} C_VEL
LIN {X 0,Y 354.789,Z 261.789,A -85,B 0,C 180,E1 -13297.9,E2 -13297.9} C_VEL
LIN {X 0,Y 354.867,Z 261.778,A -85,B 0,C 180,E1 -13301.915,E2 -13301.915} C_VEL
LIN {X 0,Y 354.923,Z 261.771,A -85,B 0,C 180,E1 -13305.989,E2 -13305.989} C_VEL
LIN {X 0,Y 354.939,Z 261.769,A -85,B 0,C 180,E1 -13309.742,E2 -13309.742} C_VEL
LIN {X 0,Y 355.091,Z 261.753,A -85,B 0,C 180,E1 -13313.187,E2 -13313.187} C_VEL
LIN {X 0,Y 355.231,Z 261.732,A -85,B 0,C 180,E1 -13317.739,E2 -13317.739} C_VEL
LIN {X 0,Y 355.344,Z 261.719,A -85,B 0,C 180,E1 -13320.007,E2 -13320.007} C_VEL
LIN {X 0,Y 355.221,Z 261.736,A -85,B 0,C 180,E1 -13322.274,E2 -13322.274} C_VEL
LIN {X 0,Y 355.1,Z 261.753,A -85,B 0,C 180,E1 -13326.826,E2 -13326.826} C_VEL
LIN {X 0,Y 354.952,Z 261.771,A -85,B 0,C 180,E1 -13330.271,E2 -13330.271} C_VEL
LIN {X 0,Y 354.943,Z 261.771,A -85,B 0,C 180,E1 -13334.024,E2 -13334.024} C_VEL
LIN {X 0,Y 354.893,Z 261.779,A -85,B 0,C 180,E1 -13338.098,E2 -13338.098} C_VEL
LIN {X 0,Y 354.819,Z 261.789,A -85,B 0,C 180,E1 -13342.113,E2 -13342.113} C_VEL
LIN {X 0,Y 354.813,Z 261.788,A -85,B 0,C 180,E1 -13345.84,E2 -13345.84} C_VEL
LIN {X 0,Y 354.804,Z 261.789,A -85,B 0,C 180,E1 -13349.689,E2 -13349.689} C_VEL
LIN {X 0,Y 354.795,Z 261.79,A -85,B 0,C 180,E1 -13352.338,E2 -13352.338} C_VEL
LIN {X 0,Y 354.828,Z 261.788,A -85,B 0,C 180,E1 -13355.702,E2 -13355.702} C_VEL
LIN {X 0,Y 354.805,Z 261.791,A -85,B 0,C 180,E1 -13356.464,E2 -13356.464} C_VEL
LIN {X 0,Y 355.315,Z 265.085,A -85,B 0,C 180,E1 -13360.753,E2 -13360.753} C_VEL
LIN {X 0,Y 355.72,Z 268.435,A -85,B 0,C 180,E1 -13364.664,E2 -13364.664} C_VEL
LIN {X 0,Y 355.85,Z 271.406,A -85,B 0,C 180,E1 -13367.819,E2 -13367.819} C_VEL
LIN {X 0,Y 355.602,Z 274.428,A -85,B 0,C 180,E1 -13370.771,E2 -13370.771} C_VEL
LIN {X 0,Y 355.208,Z 278.189,A -85,B 0,C 180,E1 -13374.221,E2 -13374.221} C_VEL
LIN {X 0,Y 354.744,Z 282.153,A -85,B 0,C 180,E1 -13377.663,E2 -13377.663} C_VEL
LIN {X 0,Y 354.318,Z 285.917,A -85,B 0,C 180,E1 -13380.787,E2 -13380.787} C_VEL
LIN {X 0,Y 353.967,Z 290.063,A -85,B 0,C 180,E1 -13384.1,E2 -13384.1} C_VEL
LIN {X 0,Y 353.76,Z 293.247,A -85,B 0,C 180,E1 -13386.589,E2 -13386.589} C_VEL
LIN {X 0,Y 353.567,Z 297.038,A -85,B 0,C 180,E1 -13389.516,E2 -13389.516} C_VEL
LIN {X 0,Y 356.712,Z 311.892,A -85,B 0,C 180,E1 -13390.292,E2 -13390.292} C_VEL
LIN {X 0,Y 358.763,Z 324.725,A -85,B 0,C 180,E1 -13391.19,E2 -13391.19} C_VEL
LIN {X 0,Y 359.66,Z 333.636,A -85,B 0,C 180,E1 -13391.929,E2 -13391.929} C_VEL
LIN {X 0,Y 358.866,Z 342.915,A -85,B 0,C 180,E1 -13392.771,E2 -13392.771} C_VEL
LIN {X 0,Y 357.867,Z 351.858,A -85,B 0,C 180,E1 -13393.749,E2 -13393.749} C_VEL
LIN {X 0,Y 356.995,Z 360.463,A -85,B 0,C 180,E1 -13394.891,E2 -13394.891} C_VEL
LIN {X 0,Y 356.206,Z 367.61,A -85,B 0,C 180,E1 -13396.014,E2 -13396.014} C_VEL
LIN {X 0,Y 355.494,Z 373.812,A -85,B 0,C 180,E1 -13397.15,E2 -13397.15} C_VEL
LIN {X 0,Y 354.695,Z 380.348,A -85,B 0,C 180,E1 -13398.572,E2 -13398.572} C_VEL
LIN {X 0,Y 354.266,Z 384.852,A -85,B 0,C 180,E1 -13399.715,E2 -13399.715} C_VEL
LIN {X 0,Y 353.742,Z 390.344,A -85,B 0,C 180,E1 -13401.431,E2 -13401.431} C_VEL
LIN {X 0,Y 353.433,Z 394.669,A -85,B 0,C 180,E1 -13403.148,E2 -13403.148} C_VEL
LIN {X 0,Y 353.303,Z 397.036,A -85,B 0,C 180,E1 -13404.292,E2 -13404.292} C_VEL
LIN {X 0,Y 353.268,Z 398.836,A -85,B 0,C 180,E1 -13405.436,E2 -13405.436} C_VEL
LIN {X 0,Y 353.177,Z 401.281,A -85,B 0,C 180,E1 -13407.719,E2 -13407.719} C_VEL
LIN {X 0,Y 353.2,Z 401.871,A -85,B 0,C 180,E1 -13408.86,E2 -13408.86} C_VEL
LIN {X 0,Y 353.2,Z 401.871,A -85,B 0,C 180,E1 -13411.14,E2 -13411.14} C_VEL
LIN {X 0,Y 353.177,Z 401.281,A -85,B 0,C 180,E1 -13412.281,E2 -13412.281} C_VEL
LIN {X 0,Y 353.266,Z 398.836,A -85,B 0,C 180,E1 -13414.564,E2 -13414.564} C_VEL
LIN {X 0,Y 353.351,Z 395.887,A -85,B 0,C 180,E1 -13416.28,E2 -13416.28} C_VEL
LIN {X 0,Y 353.63,Z 391.898,A -85,B 0,C 180,E1 -13417.997,E2 -13417.997} C_VEL
LIN {X 0,Y 354.046,Z 386.767,A -85,B 0,C 180,E1 -13419.714,E2 -13419.714} C_VEL
LIN {X 0,Y 354.593,Z 381.505,A -85,B 0,C 180,E1 -13421.142,E2 -13421.142} C_VEL
LIN {X 0,Y 355.32,Z 375.188,A -85,B 0,C 180,E1 -13422.566,E2 -13422.566} C_VEL
LIN {X 0,Y 356.031,Z 369.238,A -85,B 0,C 180,E1 -13423.702,E2 -13423.702} C_VEL
LIN {X 0,Y 356.808,Z 362.31,A -85,B 0,C 180,E1 -13424.836,E2 -13424.836} C_VEL
LIN {X 0,Y 357.592,Z 354.127,A -85,B 0,C 180,E1 -13425.971,E2 -13425.971} C_VEL
LIN {X 0,Y 358.571,Z 345.618,A -85,B 0,C 180,E1 -13426.95,E2 -13426.95} C_VEL
LIN {X 0,Y 359.435,Z 336.902,A -85,B 0,C 180,E1 -13427.789,E2 -13427.789} C_VEL
LIN {X 0,Y 359.552,Z 331.994,A -85,B 0,C 180,E1 -13428.224,E2 -13428.224} C_VEL
LIN {X 0,Y 357.937,Z 318.869,A -85,B 0,C 180,E1 -13429.24,E2 -13429.24} C_VEL
LIN {X 0,Y 355.954,Z 308.18,A -85,B 0,C 180,E1 -13429.916,E2 -13429.916} C_VEL
LIN {X 0,Y 353.575,Z 297.008,A -85,B 0,C 180,E1 -13430.507,E2 -13430.507} C_VEL
LIN {X 0,Y 353.844,Z 291.634,A -85,B 0,C 180,E1 -13434.651,E2 -13434.651} C_VEL
LIN {X 0,Y 354.06,Z 288.432,A -85,B 0,C 180,E1 -13437.164,E2 -13437.164} C_VEL
LIN {X 0,Y 354.605,Z 283.716,A -85,B 0,C 180,E1 -13441.017,E2 -13441.017} C_VEL
LIN {X 0,Y 354.965,Z 280.513,A -85,B 0,C 180,E1 -13443.734,E2 -13443.734} C_VEL
LIN {X 0,Y 355.283,Z 277.49,A -85,B 0,C 180,E1 -13446.401,E2 -13446.401} C_VEL
LIN {X 0,Y 355.635,Z 274.061,A -85,B 0,C 180,E1 -13449.576,E2 -13449.576} C_VEL
LIN {X 0,Y 355.852,Z 271.399,A -85,B 0,C 180,E1 -13452.181,E2 -13452.181} C_VEL
LIN {X 0,Y 355.713,Z 268.381,A -85,B 0,C 180,E1 -13455.337,E2 -13455.337} C_VEL
LIN {X 0,Y 355.294,Z 265.091,A -85,B 0,C 180,E1 -13459.244,E2 -13459.244} C_VEL
LIN {X 0,Y 354.926,Z 262.624,A -85,B 0,C 180,E1 -13462.376,E2 -13462.376} C_VEL
LIN {X 0,Y 354.807,Z 261.791,A -85,B 0,C 180,E1 -13463.536,E2 -13463.536} C_VEL
LIN {X 0,Y 354.824,Z 261.787,A -85,B 0,C 180,E1 -13466.312,E2 -13466.312} C_VEL
LIN {X 0,Y 354.802,Z 261.786,A -85,B 0,C 180,E1 -13468.996,E2 -13468.996} C_VEL
LIN {X 0,Y 354.807,Z 261.788,A -85,B 0,C 180,E1 -13471.61,E2 -13471.61} C_VEL
LIN {X 0,Y 354.818,Z 261.786,A -85,B 0,C 180,E1 -13475.415,E2 -13475.415} C_VEL
LIN {X 0,Y 354.829,Z 261.783,A -85,B 0,C 180,E1 -13479.108,E2 -13479.108} C_VEL
LIN {X 0,Y 354.882,Z 261.776,A -85,B 0,C 180,E1 -13482.713,E2 -13482.713} C_VEL
LIN {X 0,Y 354.951,Z 261.768,A -85,B 0,C 180,E1 -13486.249,E2 -13486.249} C_VEL
LIN {X 0,Y 354.952,Z 261.771,A -85,B 0,C 180,E1 -13489.729,E2 -13489.729} C_VEL
LIN {X 0,Y 355.1,Z 261.753,A -85,B 0,C 180,E1 -13493.174,E2 -13493.174} C_VEL
LIN {X 0,Y 355.221,Z 261.736,A -85,B 0,C 180,E1 -13497.726,E2 -13497.726} C_VEL
LIN {X 0,Y 355.344,Z 261.719,A -85,B 0,C 180,E1 -13499.993,E2 -13499.993} C_VEL
LIN {X 0,Y 355.231,Z 261.732,A -85,B 0,C 180,E1 -13502.261,E2 -13502.261} C_VEL
LIN {X 0,Y 355.091,Z 261.753,A -85,B 0,C 180,E1 -13506.813,E2 -13506.813} C_VEL
LIN {X 0,Y 354.939,Z 261.769,A -85,B 0,C 180,E1 -13510.258,E2 -13510.258} C_VEL
LIN {X 0,Y 354.923,Z 261.771,A -85,B 0,C 180,E1 -13514.011,E2 -13514.011} C_VEL
LIN {X 0,Y 354.867,Z 261.778,A -85,B 0,C 180,E1 -13518.085,E2 -13518.085} C_VEL
LIN {X 0,Y 354.789,Z 261.789,A -85,B 0,C 180,E1 -13522.1,E2 -13522.1} C_VEL
LIN {X 0,Y 354.869,Z 261.778,A -85,B 0,C 180,E1 -13525.821,E2 -13525.821} C_VEL
LIN {X 0,Y 354.772,Z 261.79,A -85,B 0,C 180,E1 -13529.676,E2 -13529.676} C_VEL
LIN {X 0,Y 354.795,Z 261.787,A -85,B 0,C 180,E1 -13533.676,E2 -13533.676} C_VEL
LIN {X 0,Y 354.761,Z 261.796,A -85,B 0,C 180,E1 -13536.453,E2 -13536.453} C_VEL
LIN {X 0,Y 354.784,Z 261.788,A -85,B 0,C 180,E1 -13539.417,E2 -13539.417} C_VEL
LIN {X 0,Y 354.801,Z 261.787,A -85,B 0,C 180,E1 -13542.871,E2 -13542.871} C_VEL
LIN {X 0,Y 354.822,Z 261.79,A -85,B 0,C 180,E1 -13546.114,E2 -13546.114} C_VEL
LIN {X 0,Y 354.809,Z 261.785,A -85,B 0,C 180,E1 -13549.183,E2 -13549.183} C_VEL
LIN {X 0,Y 354.759,Z 261.793,A -85,B 0,C 180,E1 -13552.397,E2 -13552.397} C_VEL
LIN {X 0,Y 354.76,Z 261.791,A -85,B 0,C 180,E1 -13554.936,E2 -13554.936} C_VEL
LIN {X 0,Y 354.739,Z 261.795,A -85,B 0,C 180,E1 -13558.401,E2 -13558.401} C_VEL
LIN {X 0,Y 354.797,Z 261.792,A -85,B 0,C 180,E1 -13561.615,E2 -13561.615} C_VEL
LIN {X 0,Y 354.843,Z 261.782,A -85,B 0,C 180,E1 -13564.169,E2 -13564.169} C_VEL
LIN {X 0,Y 354.833,Z 261.785,A -85,B 0,C 180,E1 -13567.894,E2 -13567.894} C_VEL
LIN {X 0,Y 354.864,Z 261.782,A -85,B 0,C 180,E1 -13571.889,E2 -13571.889} C_VEL
LIN {X 0,Y 354.89,Z 261.93,A -85,B 0,C 180,E1 -13572.331,E2 -13572.331} C_VEL
LIN {X 0,Y 355.708,Z 264.419,A -85,B 0,C 180,E1 -13572.58,E2 -13572.58} C_VEL
LIN {X 0,Y 357.601,Z 266.579,A -85,B 0,C 180,E1 -13573.036,E2 -13573.036} C_VEL
LIN {X 0,Y 358.916,Z 267.719,A -85,B 0,C 180,E1 -13573.344,E2 -13573.344} C_VEL
LIN {X 0,Y 360.975,Z 270.853,A -85,B 0,C 180,E1 -13573.898,E2 -13573.898} C_VEL
LIN {X 0,Y 363.761,Z 273.365,A -85,B 0,C 180,E1 -13574.614,E2 -13574.614} C_VEL
LIN {X 0,Y 366.171,Z 276.584,A -85,B 0,C 180,E1 -13575.303,E2 -13575.303} C_VEL
LIN {X 0,Y 369.353,Z 279.297,A -85,B 0,C 180,E1 -13576.206,E2 -13576.206} C_VEL
LIN {X 0,Y 372.29,Z 282.857,A -85,B 0,C 180,E1 -13577.153,E2 -13577.153} C_VEL
LIN {X 0,Y 375.798,Z 285.714,A -85,B 0,C 180,E1 -13578.34,E2 -13578.34} C_VEL
LIN {X 0,Y 378.642,Z 288.992,A -85,B 0,C 180,E1 -13579.439,E2 -13579.439} C_VEL
LIN {X 0,Y 381.677,Z 291.203,A -85,B 0,C 180,E1 -13580.702,E2 -13580.702} C_VEL
LIN {X 0,Y 383.274,Z 292.167,A -85,B 0,C 180,E1 -13581.432,E2 -13581.432} C_VEL
LIN {X 0,Y 385.67,Z 295.155,A -85,B 0,C 180,E1 -13582.76,E2 -13582.76} C_VEL
LIN {X 0,Y 387.806,Z 297.094,A -85,B 0,C 180,E1 -13584.167,E2 -13584.167} C_VEL
LIN {X 0,Y 389.864,Z 298.235,A -85,B 0,C 180,E1 -13585.865,E2 -13585.865} C_VEL
LIN {X 0,Y 391.49,Z 298.638,A -85,B 0,C 180,E1 -13587.942,E2 -13587.942} C_VEL
LIN {X 0,Y 391.908,Z 298.676,A -85,B 0,C 180,E1 -13588.972,E2 -13588.972} C_VEL
LIN {X 0,Y 392.046,Z 298.695,A -85,B 0,C 180,E1 -13590,E2 -13590} C_VEL
LIN {X 0,Y 391.908,Z 298.679,A -85,B 0,C 180,E1 -13591.028,E2 -13591.028} C_VEL
LIN {X 0,Y 391.49,Z 298.631,A -85,B 0,C 180,E1 -13592.058,E2 -13592.058} C_VEL
LIN {X 0,Y 389.864,Z 298.237,A -85,B 0,C 180,E1 -13594.135,E2 -13594.135} C_VEL
LIN {X 0,Y 387.806,Z 297.093,A -85,B 0,C 180,E1 -13595.833,E2 -13595.833} C_VEL
LIN {X 0,Y 385.652,Z 295.134,A -85,B 0,C 180,E1 -13597.252,E2 -13597.252} C_VEL
LIN {X 0,Y 383.174,Z 292.023,A -85,B 0,C 180,E1 -13598.62,E2 -13598.62} C_VEL
LIN {X 0,Y 379.709,Z 289.903,A -85,B 0,C 180,E1 -13600.127,E2 -13600.127} C_VEL
LIN {X 0,Y 376.741,Z 286.924,A -85,B 0,C 180,E1 -13601.311,E2 -13601.311} C_VEL
LIN {X 0,Y 375.158,Z 285.021,A -85,B 0,C 180,E1 -13601.892,E2 -13601.892} C_VEL
LIN {X 0,Y 371.709,Z 282.316,A -85,B 0,C 180,E1 -13603.027,E2 -13603.027} C_VEL
LIN {X 0,Y 368.721,Z 278.583,A -85,B 0,C 180,E1 -13603.984,E2 -13603.984} C_VEL
LIN {X 0,Y 365.75,Z 276.134,A -85,B 0,C 180,E1 -13604.817,E2 -13604.817} C_VEL
LIN {X 0,Y 363.068,Z 272.616,A -85,B 0,C 180,E1 -13605.568,E2 -13605.568} C_VEL
LIN {X 0,Y 360.339,Z 270.075,A -85,B 0,C 180,E1 -13606.273,E2 -13606.273} C_VEL
LIN {X 0,Y 358.397,Z 267.101,A -85,B 0,C 180,E1 -13606.783,E2 -13606.783} C_VEL
LIN {X 0,Y 356.11,Z 265.034,A -85,B 0,C 180,E1 -13607.318,E2 -13607.318} C_VEL
LIN {X 0,Y 354.953,Z 262.431,A -85,B 0,C 180,E1 -13607.64,E2 -13607.64} C_VEL
LIN {X 0,Y 354.866,Z 261.782,A -85,B 0,C 180,E1 -13607.696,E2 -13607.696} C_VEL
LIN {X 0,Y 354.83,Z 261.783,A -85,B 0,C 180,E1 -13611.45,E2 -13611.45} C_VEL
LIN {X 0,Y 354.819,Z 261.788,A -85,B 0,C 180,E1 -13614.579,E2 -13614.579} C_VEL
LIN {X 0,Y 354.829,Z 261.783,A -85,B 0,C 180,E1 -13617.1,E2 -13617.1} C_VEL
LIN {X 0,Y 354.8,Z 261.787,A -85,B 0,C 180,E1 -13619.683,E2 -13619.683} C_VEL
LIN {X 0,Y 354.754,Z 261.794,A -85,B 0,C 180,E1 -13623.707,E2 -13623.707} C_VEL
LIN {X 0,Y 354.748,Z 261.795,A -85,B 0,C 180,E1 -13626.464,E2 -13626.464} C_VEL
LIN {X 0,Y 354.776,Z 261.79,A -85,B 0,C 180,E1 -13629.429,E2 -13629.429} C_VEL
LIN {X 0,Y 354.796,Z 261.787,A -85,B 0,C 180,E1 -13632.882,E2 -13632.882} C_VEL
LIN {X 0,Y 354.824,Z 261.787,A -85,B 0,C 180,E1 -13636.125,E2 -13636.125} C_VEL
LIN {X 0,Y 354.787,Z 261.786,A -85,B 0,C 180,E1 -13639.567,E2 -13639.567} C_VEL
LIN {X 0,Y 354.761,Z 261.796,A -85,B 0,C 180,E1 -13643.547,E2 -13643.547} C_VEL
LIN {X 0,Y 354.777,Z 261.789,A -85,B 0,C 180,E1 -13644.503,E2 -13644.503} C_VEL
LIN {X 0,Y 354.087,Z 261.879,A -85,B 0,C 180,E1 -13645.45,E2 -13645.45} C_VEL
LIN {X 0,Y 351.193,Z 262.236,A -85,B 0,C 180,E1 -13646.99,E2 -13646.99} C_VEL
LIN {X 0,Y 348.773,Z 262.538,A -85,B 0,C 180,E1 -13648.236,E2 -13648.236} C_VEL
LIN {X 0,Y 347.766,Z 262.665,A -85,B 0,C 180,E1 -13649.201,E2 -13649.201} C_VEL
LIN {X 0,Y 347.701,Z 262.674,A -85,B 0,C 180,E1 -13649.528,E2 -13649.528} C_VEL
LIN {X 0,Y 347.801,Z 262.662,A -85,B 0,C 180,E1 -13653.615,E2 -13653.615} C_VEL
LIN {X 0,Y 347.757,Z 262.664,A -85,B 0,C 180,E1 -13656.169,E2 -13656.169} C_VEL
LIN {X 0,Y 347.761,Z 262.663,A -85,B 0,C 180,E1 -13659.915,E2 -13659.915} C_VEL
LIN {X 0,Y 347.81,Z 262.659,A -85,B 0,C 180,E1 -13663.575,E2 -13663.575} C_VEL
LIN {X 0,Y 347.871,Z 262.655,A -85,B 0,C 180,E1 -13667.168,E2 -13667.168} C_VEL
LIN {X 0,Y 347.92,Z 262.646,A -85,B 0,C 180,E1 -13670.708,E2 -13670.708} C_VEL
LIN {X 0,Y 348.058,Z 262.631,A -85,B 0,C 180,E1 -13673.049,E2 -13673.049} C_VEL
LIN {X 0,Y 348.193,Z 262.608,A -85,B 0,C 180,E1 -13677.693,E2 -13677.693} C_VEL
LIN {X 0,Y 348.294,Z 262.596,A -85,B 0,C 180,E1 -13680.007,E2 -13680.007} C_VEL
LIN {X 0,Y 348.183,Z 262.613,A -85,B 0,C 180,E1 -13682.32,E2 -13682.32} C_VEL
LIN {X 0,Y 348.068,Z 262.627,A -85,B 0,C 180,E1 -13686.965,E2 -13686.965} C_VEL
LIN {X 0,Y 347.893,Z 262.653,A -85,B 0,C 180,E1 -13690.482,E2 -13690.482} C_VEL
LIN {X 0,Y 347.9,Z 262.649,A -85,B 0,C 180,E1 -13694.156,E2 -13694.156} C_VEL
LIN {X 0,Y 347.832,Z 262.66,A -85,B 0,C 180,E1 -13698.265,E2 -13698.265} C_VEL
LIN {X 0,Y 347.771,Z 262.663,A -85,B 0,C 180,E1 -13701.631,E2 -13701.631} C_VEL
LIN {X 0,Y 347.751,Z 262.665,A -85,B 0,C 180,E1 -13705.119,E2 -13705.119} C_VEL
LIN {X 0,Y 347.743,Z 262.668,A -85,B 0,C 180,E1 -13707.705,E2 -13707.705} C_VEL
LIN {X 0,Y 347.746,Z 262.668,A -85,B 0,C 180,E1 -13710.354,E2 -13710.354} C_VEL
LIN {X 0,Y 347.758,Z 262.67,A -85,B 0,C 180,E1 -13714.048,E2 -13714.048} C_VEL
LIN {X 0,Y 347.777,Z 262.667,A -85,B 0,C 180,E1 -13716.069,E2 -13716.069} C_VEL
LIN {X 0,Y 348.213,Z 265.739,A -85,B 0,C 180,E1 -13720.236,E2 -13720.236} C_VEL
LIN {X 0,Y 348.564,Z 268.418,A -85,B 0,C 180,E1 -13723.461,E2 -13723.461} C_VEL
LIN {X 0,Y 348.777,Z 269.905,A -85,B 0,C 180,E1 -13725.151,E2 -13725.151} C_VEL
LIN {X 0,Y 348.791,Z 272.858,A -85,B 0,C 180,E1 -13728.324,E2 -13728.324} C_VEL
LIN {X 0,Y 348.439,Z 276.484,A -85,B 0,C 180,E1 -13731.878,E2 -13731.878} C_VEL
LIN {X 0,Y 348.173,Z 278.952,A -85,B 0,C 180,E1 -13734.171,E2 -13734.171} C_VEL
LIN {X 0,Y 347.643,Z 283.417,A -85,B 0,C 180,E1 -13738.119,E2 -13738.119} C_VEL
LIN {X 0,Y 347.231,Z 286.76,A -85,B 0,C 180,E1 -13740.938,E2 -13740.938} C_VEL
LIN {X 0,Y 346.822,Z 291.499,A -85,B 0,C 180,E1 -13744.816,E2 -13744.816} C_VEL
LIN {X 0,Y 346.506,Z 296.265,A -85,B 0,C 180,E1 -13748.588,E2 -13748.588} C_VEL
LIN {X 0,Y 346.503,Z 296.89,A -85,B 0,C 180,E1 -13749.094,E2 -13749.094} C_VEL
LIN {X 0,Y 348.794,Z 307.246,A -85,B 0,C 180,E1 -13749.626,E2 -13749.626} C_VEL
LIN {X 0,Y 350.617,Z 316.928,A -85,B 0,C 180,E1 -13750.24,E2 -13750.24} C_VEL
LIN {X 0,Y 351.866,Z 325.343,A -85,B 0,C 180,E1 -13750.869,E2 -13750.869} C_VEL
LIN {X 0,Y 352.782,Z 333.437,A -85,B 0,C 180,E1 -13751.564,E2 -13751.564} C_VEL
LIN {X 0,Y 352.078,Z 342.72,A -85,B 0,C 180,E1 -13752.428,E2 -13752.428} C_VEL
LIN {X 0,Y 351.016,Z 351.662,A -85,B 0,C 180,E1 -13753.423,E2 -13753.423} C_VEL
LIN {X 0,Y 350.136,Z 360.118,A -85,B 0,C 180,E1 -13754.565,E2 -13754.565} C_VEL
LIN {X 0,Y 349.268,Z 367.414,A -85,B 0,C 180,E1 -13755.73,E2 -13755.73} C_VEL
LIN {X 0,Y 348.545,Z 373.617,A -85,B 0,C 180,E1 -13756.889,E2 -13756.889} C_VEL
LIN {X 0,Y 347.706,Z 380.153,A -85,B 0,C 180,E1 -13758.339,E2 -13758.339} C_VEL
LIN {X 0,Y 347.27,Z 384.657,A -85,B 0,C 180,E1 -13759.506,E2 -13759.506} C_VEL
LIN {X 0,Y 346.697,Z 390.148,A -85,B 0,C 180,E1 -13761.255,E2 -13761.255} C_VEL
LIN {X 0,Y 346.36,Z 394.474,A -85,B 0,C 180,E1 -13763.007,E2 -13763.007} C_VEL
LIN {X 0,Y 346.219,Z 396.841,A -85,B 0,C 180,E1 -13764.175,E2 -13764.175} C_VEL
LIN {X 0,Y 346.167,Z 398.641,A -85,B 0,C 180,E1 -13765.342,E2 -13765.342} C_VEL
LIN {X 0,Y 346.088,Z 401.087,A -85,B 0,C 180,E1 -13767.672,E2 -13767.672} C_VEL
LIN {X 0,Y 346.1,Z 401.676,A -85,B 0,C 180,E1 -13768.836,E2 -13768.836} C_VEL
LIN {X 0,Y 346.1,Z 401.676,A -85,B 0,C 180,E1 -13771.164,E2 -13771.164} C_VEL
LIN {X 0,Y 346.088,Z 401.087,A -85,B 0,C 180,E1 -13772.328,E2 -13772.328} C_VEL
LIN {X 0,Y 346.165,Z 398.641,A -85,B 0,C 180,E1 -13774.658,E2 -13774.658} C_VEL
LIN {X 0,Y 346.279,Z 395.692,A -85,B 0,C 180,E1 -13776.408,E2 -13776.408} C_VEL
LIN {X 0,Y 346.569,Z 391.703,A -85,B 0,C 180,E1 -13778.161,E2 -13778.161} C_VEL
LIN {X 0,Y 347.031,Z 386.572,A -85,B 0,C 180,E1 -13779.912,E2 -13779.912} C_VEL
LIN {X 0,Y 347.575,Z 381.309,A -85,B 0,C 180,E1 -13781.37,E2 -13781.37} C_VEL
LIN {X 0,Y 348.36,Z 374.993,A -85,B 0,C 180,E1 -13782.822,E2 -13782.822} C_VEL
LIN {X 0,Y 349.094,Z 369.042,A -85,B 0,C 180,E1 -13783.98,E2 -13783.98} C_VEL
LIN {X 0,Y 350.013,Z 361.189,A -85,B 0,C 180,E1 -13785.274,E2 -13785.274} C_VEL
LIN {X 0,Y 350.864,Z 352.796,A -85,B 0,C 180,E1 -13786.435,E2 -13786.435} C_VEL
LIN {X 0,Y 351.897,Z 344.07,A -85,B 0,C 180,E1 -13787.432,E2 -13787.432} C_VEL
LIN {X 0,Y 352.783,Z 335.074,A -85,B 0,C 180,E1 -13788.286,E2 -13788.286} C_VEL
LIN {X 0,Y 352.079,Z 326.827,A -85,B 0,C 180,E1 -13789.009,E2 -13789.009} C_VEL
LIN {X 0,Y 350.827,Z 318.094,A -85,B 0,C 180,E1 -13789.679,E2 -13789.679} C_VEL
LIN {X 0,Y 348.793,Z 307.257,A -85,B 0,C 180,E1 -13790.374,E2 -13790.374} C_VEL
LIN {X 0,Y 346.495,Z 296.878,A -85,B 0,C 180,E1 -13790.916,E2 -13790.916} C_VEL
LIN {X 0,Y 346.743,Z 292.711,A -85,B 0,C 180,E1 -13794.196,E2 -13794.196} C_VEL
LIN {X 0,Y 347.053,Z 288.313,A -85,B 0,C 180,E1 -13797.759,E2 -13797.759} C_VEL
LIN {X 0,Y 347.623,Z 283.611,A -85,B 0,C 180,E1 -13801.711,E2 -13801.711} C_VEL
LIN {X 0,Y 347.971,Z 280.493,A -85,B 0,C 180,E1 -13804.437,E2 -13804.437} C_VEL
LIN {X 0,Y 348.436,Z 276.484,A -85,B 0,C 180,E1 -13808.121,E2 -13808.121} C_VEL
LIN {X 0,Y 348.79,Z 272.739,A -85,B 0,C 180,E1 -13811.789,E2 -13811.789} C_VEL
LIN {X 0,Y 348.775,Z 269.842,A -85,B 0,C 180,E1 -13814.85,E2 -13814.85} C_VEL
LIN {X 0,Y 348.369,Z 266.915,A -85,B 0,C 180,E1 -13818.281,E2 -13818.281} C_VEL
LIN {X 0,Y 347.94,Z 264.061,A -85,B 0,C 180,E1 -13821.974,E2 -13821.974} C_VEL
LIN {X 0,Y 347.797,Z 262.666,A -85,B 0,C 180,E1 -13824.12,E2 -13824.12} C_VEL
LIN {X 0,Y 347.747,Z 262.671,A -85,B 0,C 180,E1 -13828.082,E2 -13828.082} C_VEL
LIN {X 0,Y 347.753,Z 262.664,A -85,B 0,C 180,E1 -13830.98,E2 -13830.98} C_VEL
LIN {X 0,Y 347.752,Z 262.668,A -85,B 0,C 180,E1 -13833.595,E2 -13833.595} C_VEL
LIN {X 0,Y 347.764,Z 262.666,A -85,B 0,C 180,E1 -13836.154,E2 -13836.154} C_VEL
LIN {X 0,Y 347.801,Z 262.663,A -85,B 0,C 180,E1 -13839.903,E2 -13839.903} C_VEL
LIN {X 0,Y 347.833,Z 262.66,A -85,B 0,C 180,E1 -13843.562,E2 -13843.562} C_VEL
LIN {X 0,Y 347.889,Z 262.65,A -85,B 0,C 180,E1 -13847.154,E2 -13847.154} C_VEL
LIN {X 0,Y 347.932,Z 262.642,A -85,B 0,C 180,E1 -13850.694,E2 -13850.694} C_VEL
LIN {X 0,Y 348.068,Z 262.627,A -85,B 0,C 180,E1 -13853.035,E2 -13853.035} C_VEL
LIN {X 0,Y 348.183,Z 262.613,A -85,B 0,C 180,E1 -13857.68,E2 -13857.68} C_VEL
LIN {X 0,Y 348.294,Z 262.596,A -85,B 0,C 180,E1 -13859.993,E2 -13859.993} C_VEL
LIN {X 0,Y 348.193,Z 262.608,A -85,B 0,C 180,E1 -13862.307,E2 -13862.307} C_VEL
LIN {X 0,Y 348.058,Z 262.631,A -85,B 0,C 180,E1 -13866.951,E2 -13866.951} C_VEL
LIN {X 0,Y 347.879,Z 262.65,A -85,B 0,C 180,E1 -13870.468,E2 -13870.468} C_VEL
LIN {X 0,Y 347.88,Z 262.648,A -85,B 0,C 180,E1 -13874.143,E2 -13874.143} C_VEL
LIN {X 0,Y 347.806,Z 262.659,A -85,B 0,C 180,E1 -13878.252,E2 -13878.252} C_VEL
LIN {X 0,Y 347.742,Z 262.666,A -85,B 0,C 180,E1 -13881.619,E2 -13881.619} C_VEL
LIN {X 0,Y 347.782,Z 262.662,A -85,B 0,C 180,E1 -13885.102,E2 -13885.102} C_VEL
LIN {X 0,Y 347.771,Z 262.662,A -85,B 0,C 180,E1 -13887.688,E2 -13887.688} C_VEL
LIN {X 0,Y 347.712,Z 262.67,A -85,B 0,C 180,E1 -13891.693,E2 -13891.693} C_VEL
LIN {X 0,Y 347.708,Z 262.675,A -85,B 0,C 180,E1 -13894.457,E2 -13894.457} C_VEL
LIN {X 0,Y 347.736,Z 262.669,A -85,B 0,C 180,E1 -13897.982,E2 -13897.982} C_VEL
LIN {X 0,Y 347.745,Z 262.666,A -85,B 0,C 180,E1 -13901.603,E2 -13901.603} C_VEL
LIN {X 0,Y 347.787,Z 262.66,A -85,B 0,C 180,E1 -13905,E2 -13905} C_VEL
LIN {X 0,Y 347.738,Z 262.669,A -85,B 0,C 180,E1 -13908.385,E2 -13908.385} C_VEL
LIN {X 0,Y 347.726,Z 262.673,A -85,B 0,C 180,E1 -13912.006,E2 -13912.006} C_VEL
LIN {X 0,Y 347.692,Z 262.675,A -85,B 0,C 180,E1 -13915.531,E2 -13915.531} C_VEL
LIN {X 0,Y 347.71,Z 262.675,A -85,B 0,C 180,E1 -13919.649,E2 -13919.649} C_VEL
LIN {X 0,Y 347.797,Z 262.659,A -85,B 0,C 180,E1 -13922.741,E2 -13922.741} C_VEL
LIN {X 0,Y 347.76,Z 262.665,A -85,B 0,C 180,E1 -13926.16,E2 -13926.16} C_VEL
LIN {X 0,Y 347.785,Z 262.665,A -85,B 0,C 180,E1 -13929.908,E2 -13929.908} C_VEL
LIN {X 0,Y 347.794,Z 262.697,A -85,B 0,C 180,E1 -13931.022,E2 -13931.022} C_VEL
LIN {X 0,Y 348.72,Z 265.344,A -85,B 0,C 180,E1 -13931.271,E2 -13931.271} C_VEL
LIN {X 0,Y 350.781,Z 267.57,A -85,B 0,C 180,E1 -13931.721,E2 -13931.721} C_VEL
LIN {X 0,Y 351.478,Z 268.274,A -85,B 0,C 180,E1 -13931.874,E2 -13931.874} C_VEL
LIN {X 0,Y 353.527,Z 271.421,A -85,B 0,C 180,E1 -13932.358,E2 -13932.358} C_VEL
LIN {X 0,Y 356.091,Z 274.022,A -85,B 0,C 180,E1 -13932.964,E2 -13932.964} C_VEL
LIN {X 0,Y 358.673,Z 277.342,A -85,B 0,C 180,E1 -13933.602,E2 -13933.602} C_VEL
LIN {X 0,Y 361.101,Z 279.595,A -85,B 0,C 180,E1 -13934.223,E2 -13934.223} C_VEL
LIN {X 0,Y 364.212,Z 283.243,A -85,B 0,C 180,E1 -13935.055,E2 -13935.055} C_VEL
LIN {X 0,Y 367.257,Z 285.912,A -85,B 0,C 180,E1 -13935.908,E2 -13935.908} C_VEL
LIN {X 0,Y 370.226,Z 289.3,A -85,B 0,C 180,E1 -13936.833,E2 -13936.833} C_VEL
LIN {X 0,Y 373.848,Z 292.173,A -85,B 0,C 180,E1 -13938,E2 -13938} C_VEL
LIN {X 0,Y 376.832,Z 295.531,A -85,B 0,C 180,E1 -13939.115,E2 -13939.115} C_VEL
LIN {X 0,Y 380.395,Z 298.115,A -85,B 0,C 180,E1 -13940.551,E2 -13940.551} C_VEL
LIN {X 0,Y 381.932,Z 299.091,A -85,B 0,C 180,E1 -13941.235,E2 -13941.235} C_VEL
LIN {X 0,Y 384.561,Z 302.156,A -85,B 0,C 180,E1 -13942.65,E2 -13942.65} C_VEL
LIN {X 0,Y 386.894,Z 304.156,A -85,B 0,C 180,E1 -13944.153,E2 -13944.153} C_VEL
LIN {X 0,Y 388.977,Z 305.256,A -85,B 0,C 180,E1 -13945.856,E2 -13945.856} C_VEL
LIN {X 0,Y 389.935,Z 305.5,A -85,B 0,C 180,E1 -13946.901,E2 -13946.901} C_VEL
LIN {X 0,Y 390.618,Z 305.683,A -85,B 0,C 180,E1 -13947.938,E2 -13947.938} C_VEL
LIN {X 0,Y 391.042,Z 305.704,A -85,B 0,C 180,E1 -13948.97,E2 -13948.97} C_VEL
LIN {X 0,Y 391.182,Z 305.73,A -85,B 0,C 180,E1 -13950,E2 -13950} C_VEL
LIN {X 0,Y 391.042,Z 305.708,A -85,B 0,C 180,E1 -13951.03,E2 -13951.03} C_VEL
LIN {X 0,Y 390.618,Z 305.677,A -85,B 0,C 180,E1 -13952.062,E2 -13952.062} C_VEL
LIN {X 0,Y 389.479,Z 305.421,A -85,B 0,C 180,E1 -13953.657,E2 -13953.657} C_VEL
LIN {X 0,Y 387.603,Z 304.597,A -85,B 0,C 180,E1 -13955.332,E2 -13955.332} C_VEL
LIN {X 0,Y 385.259,Z 302.877,A -85,B 0,C 180,E1 -13956.919,E2 -13956.919} C_VEL
LIN {X 0,Y 382.533,Z 299.9,A -85,B 0,C 180,E1 -13958.452,E2 -13958.452} C_VEL
LIN {X 0,Y 381.447,Z 298.617,A -85,B 0,C 180,E1 -13959.001,E2 -13959.001} C_VEL
LIN {X 0,Y 378.195,Z 296.674,A -85,B 0,C 180,E1 -13960.354,E2 -13960.354} C_VEL
LIN {X 0,Y 374.812,Z 293.406,A -85,B 0,C 180,E1 -13961.642,E2 -13961.642} C_VEL
LIN {X 0,Y 373.177,Z 291.563,A -85,B 0,C 180,E1 -13962.232,E2 -13962.232} C_VEL
LIN {X 0,Y 369.546,Z 288.681,A -85,B 0,C 180,E1 -13963.38,E2 -13963.38} C_VEL
LIN {X 0,Y 366.374,Z 284.986,A -85,B 0,C 180,E1 -13964.348,E2 -13964.348} C_VEL
LIN {X 0,Y 363.049,Z 282.079,A -85,B 0,C 180,E1 -13965.251,E2 -13965.251} C_VEL
LIN {X 0,Y 360.46,Z 278.876,A -85,B 0,C 180,E1 -13965.949,E2 -13965.949} C_VEL
LIN {X 0,Y 357.322,Z 275.854,A -85,B 0,C 180,E1 -13966.722,E2 -13966.722} C_VEL
LIN {X 0,Y 355.351,Z 273.126,A -85,B 0,C 180,E1 -13967.217,E2 -13967.217} C_VEL
LIN {X 0,Y 352.693,Z 270.415,A -85,B 0,C 180,E1 -13967.829,E2 -13967.829} C_VEL
LIN {X 0,Y 351.065,Z 267.759,A -85,B 0,C 180,E1 -13968.22,E2 -13968.22} C_VEL
LIN {X 0,Y 348.881,Z 265.652,A -85,B 0,C 180,E1 -13968.69,E2 -13968.69} C_VEL
LIN {X 0,Y 347.921,Z 263.448,A -85,B 0,C 180,E1 -13968.932,E2 -13968.932} C_VEL
LIN {X 0,Y 347.783,Z 262.665,A -85,B 0,C 180,E1 -13969.017,E2 -13969.017} C_VEL
LIN {X 0,Y 347.782,Z 262.666,A -85,B 0,C 180,E1 -13972.578,E2 -13972.578} C_VEL
LIN {X 0,Y 347.777,Z 262.667,A -85,B 0,C 180,E1 -13976.396,E2 -13976.396} C_VEL
LIN {X 0,Y 347.755,Z 262.665,A -85,B 0,C 180,E1 -13979.676,E2 -13979.676} C_VEL
LIN {X 0,Y 347.68,Z 262.673,A -85,B 0,C 180,E1 -13983.077,E2 -13983.077} C_VEL
LIN {X 0,Y 347.72,Z 262.674,A -85,B 0,C 180,E1 -13986.07,E2 -13986.07} C_VEL
LIN {X 0,Y 347.738,Z 262.67,A -85,B 0,C 180,E1 -13989.84,E2 -13989.84} C_VEL
LIN {X 0,Y 347.774,Z 262.663,A -85,B 0,C 180,E1 -13993.399,E2 -13993.399} C_VEL
LIN {X 0,Y 347.775,Z 262.661,A -85,B 0,C 180,E1 -13996.676,E2 -13996.676} C_VEL
LIN {X 0,Y 347.746,Z 262.667,A -85,B 0,C 180,E1 -14000.172,E2 -14000.172} C_VEL
LIN {X 0,Y 347.751,Z 262.666,A -85,B 0,C 180,E1 -14004.131,E2 -14004.131} C_VEL
LIN {X 0,Y 347.706,Z 262.671,A -85,B 0,C 180,E1 -14008.093,E2 -14008.093} C_VEL
LIN {X 0,Y 347.701,Z 262.674,A -85,B 0,C 180,E1 -14009.528,E2 -14009.528} C_VEL
LIN {X 0,Y 347.085,Z 262.757,A -85,B 0,C 180,E1 -14010.496,E2 -14010.496} C_VEL
LIN {X 0,Y 344.272,Z 263.105,A -85,B 0,C 180,E1 -14012.071,E2 -14012.071} C_VEL
LIN {X 0,Y 341.859,Z 263.404,A -85,B 0,C 180,E1 -14013.346,E2 -14013.346} C_VEL
LIN {X 0,Y 340.818,Z 263.528,A -85,B 0,C 180,E1 -14014.332,E2 -14014.332} C_VEL
LIN {X 0,Y 340.732,Z 263.539,A -85,B 0,C 180,E1 -14014.667,E2 -14014.667} C_VEL
LIN {X 0,Y 340.716,Z 263.541,A -85,B 0,C 180,E1 -14018.214,E2 -14018.214} C_VEL
LIN {X 0,Y 340.77,Z 263.534,A -85,B 0,C 180,E1 -14021.988,E2 -14021.988} C_VEL
LIN {X 0,Y 340.833,Z 263.527,A -85,B 0,C 180,E1 -14025.724,E2 -14025.724} C_VEL
LIN {X 0,Y 340.831,Z 263.529,A -85,B 0,C 180,E1 -14029.313,E2 -14029.313} C_VEL
LIN {X 0,Y 341.027,Z 263.508,A -85,B 0,C 180,E1 -14032.905,E2 -14032.905} C_VEL
LIN {X 0,Y 341.155,Z 263.483,A -85,B 0,C 180,E1 -14037.646,E2 -14037.646} C_VEL
LIN {X 0,Y 341.246,Z 263.473,A -85,B 0,C 180,E1 -14040.007,E2 -14040.007} C_VEL
LIN {X 0,Y 341.12,Z 263.493,A -85,B 0,C 180,E1 -14042.368,E2 -14042.368} C_VEL
LIN {X 0,Y 341.015,Z 263.505,A -85,B 0,C 180,E1 -14047.11,E2 -14047.11} C_VEL
LIN {X 0,Y 340.845,Z 263.529,A -85,B 0,C 180,E1 -14050.701,E2 -14050.701} C_VEL
LIN {X 0,Y 340.865,Z 263.528,A -85,B 0,C 180,E1 -14054.331,E2 -14054.331} C_VEL
LIN {X 0,Y 340.789,Z 263.536,A -85,B 0,C 180,E1 -14058.446,E2 -14058.446} C_VEL
LIN {X 0,Y 340.723,Z 263.542,A -85,B 0,C 180,E1 -14061.847,E2 -14061.847} C_VEL
LIN {X 0,Y 340.721,Z 263.541,A -85,B 0,C 180,E1 -14064.83,E2 -14064.83} C_VEL
LIN {X 0,Y 340.69,Z 263.548,A -85,B 0,C 180,E1 -14068.33,E2 -14068.33} C_VEL
LIN {X 0,Y 340.702,Z 263.544,A -85,B 0,C 180,E1 -14071.05,E2 -14071.05} C_VEL
LIN {X 0,Y 340.726,Z 263.543,A -85,B 0,C 180,E1 -14075.284,E2 -14075.284} C_VEL
LIN {X 0,Y 340.818,Z 264.228,A -85,B 0,C 180,E1 -14076.733,E2 -14076.733} C_VEL
LIN {X 0,Y 341.208,Z 266.913,A -85,B 0,C 180,E1 -14080.352,E2 -14080.352} C_VEL
LIN {X 0,Y 341.588,Z 269.858,A -85,B 0,C 180,E1 -14083.938,E2 -14083.938} C_VEL
LIN {X 0,Y 341.741,Z 271.675,A -85,B 0,C 180,E1 -14086.043,E2 -14086.043} C_VEL
LIN {X 0,Y 341.695,Z 274.302,A -85,B 0,C 180,E1 -14088.84,E2 -14088.84} C_VEL
LIN {X 0,Y 341.387,Z 277.337,A -85,B 0,C 180,E1 -14091.86,E2 -14091.86} C_VEL
LIN {X 0,Y 340.909,Z 281.275,A -85,B 0,C 180,E1 -14095.557,E2 -14095.557} C_VEL
LIN {X 0,Y 340.444,Z 285.067,A -85,B 0,C 180,E1 -14098.93,E2 -14098.93} C_VEL
LIN {X 0,Y 339.914,Z 289.771,A -85,B 0,C 180,E1 -14102.944,E2 -14102.944} C_VEL
LIN {X 0,Y 339.697,Z 292.953,A -85,B 0,C 180,E1 -14105.558,E2 -14105.558} C_VEL
LIN {X 0,Y 339.418,Z 296.714,A -85,B 0,C 180,E1 -14108.629,E2 -14108.629} C_VEL
LIN {X 0,Y 342.561,Z 310.77,A -85,B 0,C 180,E1 -14109.405,E2 -14109.405} C_VEL
LIN {X 0,Y 344.708,Z 323.349,A -85,B 0,C 180,E1 -14110.318,E2 -14110.318} C_VEL
LIN {X 0,Y 345.848,Z 333.236,A -85,B 0,C 180,E1 -14111.18,E2 -14111.18} C_VEL
LIN {X 0,Y 345.671,Z 339.756,A -85,B 0,C 180,E1 -14111.785,E2 -14111.785} C_VEL
LIN {X 0,Y 344.353,Z 350.333,A -85,B 0,C 180,E1 -14112.94,E2 -14112.94} C_VEL
LIN {X 0,Y 343.282,Z 359.711,A -85,B 0,C 180,E1 -14114.215,E2 -14114.215} C_VEL
LIN {X 0,Y 342.34,Z 367.218,A -85,B 0,C 180,E1 -14115.435,E2 -14115.435} C_VEL
LIN {X 0,Y 341.612,Z 373.422,A -85,B 0,C 180,E1 -14116.618,E2 -14116.618} C_VEL
LIN {X 0,Y 340.729,Z 379.957,A -85,B 0,C 180,E1 -14118.097,E2 -14118.097} C_VEL
LIN {X 0,Y 340.257,Z 384.461,A -85,B 0,C 180,E1 -14119.287,E2 -14119.287} C_VEL
LIN {X 0,Y 339.641,Z 389.952,A -85,B 0,C 180,E1 -14121.072,E2 -14121.072} C_VEL
LIN {X 0,Y 339.291,Z 394.279,A -85,B 0,C 180,E1 -14122.861,E2 -14122.861} C_VEL
LIN {X 0,Y 339.15,Z 396.745,A -85,B 0,C 180,E1 -14124.117,E2 -14124.117} C_VEL
LIN {X 0,Y 339.07,Z 399.835,A -85,B 0,C 180,E1 -14126.435,E2 -14126.435} C_VEL
LIN {X 0,Y 339.003,Z 400.892,A -85,B 0,C 180,E1 -14127.624,E2 -14127.624} C_VEL
LIN {X 0,Y 339.005,Z 401.481,A -85,B 0,C 180,E1 -14128.812,E2 -14128.812} C_VEL
LIN {X 0,Y 339.005,Z 401.481,A -85,B 0,C 180,E1 -14131.188,E2 -14131.188} C_VEL
LIN {X 0,Y 339.003,Z 400.892,A -85,B 0,C 180,E1 -14132.376,E2 -14132.376} C_VEL
LIN {X 0,Y 339.069,Z 398.446,A -85,B 0,C 180,E1 -14134.756,E2 -14134.756} C_VEL
LIN {X 0,Y 339.194,Z 395.496,A -85,B 0,C 180,E1 -14136.543,E2 -14136.543} C_VEL
LIN {X 0,Y 339.528,Z 391.507,A -85,B 0,C 180,E1 -14138.331,E2 -14138.331} C_VEL
LIN {X 0,Y 340.008,Z 386.376,A -85,B 0,C 180,E1 -14140.119,E2 -14140.119} C_VEL
LIN {X 0,Y 340.583,Z 381.113,A -85,B 0,C 180,E1 -14141.606,E2 -14141.606} C_VEL
LIN {X 0,Y 341.414,Z 374.797,A -85,B 0,C 180,E1 -14143.087,E2 -14143.087} C_VEL
LIN {X 0,Y 342.165,Z 368.846,A -85,B 0,C 180,E1 -14144.269,E2 -14144.269} C_VEL
LIN {X 0,Y 343.033,Z 361.919,A -85,B 0,C 180,E1 -14145.446,E2 -14145.446} C_VEL
LIN {X 0,Y 343.898,Z 353.735,A -85,B 0,C 180,E1 -14146.625,E2 -14146.625} C_VEL
LIN {X 0,Y 344.969,Z 345.227,A -85,B 0,C 180,E1 -14147.64,E2 -14147.64} C_VEL
LIN {X 0,Y 345.902,Z 336.511,A -85,B 0,C 180,E1 -14148.509,E2 -14148.509} C_VEL
LIN {X 0,Y 345.336,Z 328.477,A -85,B 0,C 180,E1 -14149.253,E2 -14149.253} C_VEL
LIN {X 0,Y 344.064,Z 319.217,A -85,B 0,C 180,E1 -14150.003,E2 -14150.003} C_VEL
LIN {X 0,Y 341.982,Z 308.055,A -85,B 0,C 180,E1 -14150.753,E2 -14150.753} C_VEL
LIN {X 0,Y 339.525,Z 297.683,A -85,B 0,C 180,E1 -14151.324,E2 -14151.324} C_VEL
LIN {X 0,Y 339.415,Z 296.688,A -85,B 0,C 180,E1 -14151.393,E2 -14151.393} C_VEL
LIN {X 0,Y 339.697,Z 292.916,A -85,B 0,C 180,E1 -14154.442,E2 -14154.442} C_VEL
LIN {X 0,Y 340.038,Z 288.193,A -85,B 0,C 180,E1 -14158.383,E2 -14158.383} C_VEL
LIN {X 0,Y 340.447,Z 285.055,A -85,B 0,C 180,E1 -14161.069,E2 -14161.069} C_VEL
LIN {X 0,Y 340.92,Z 281.269,A -85,B 0,C 180,E1 -14164.446,E2 -14164.446} C_VEL
LIN {X 0,Y 341.384,Z 277.332,A -85,B 0,C 180,E1 -14168.14,E2 -14168.14} C_VEL
LIN {X 0,Y 341.695,Z 274.288,A -85,B 0,C 180,E1 -14171.16,E2 -14171.16} C_VEL
LIN {X 0,Y 341.75,Z 271.302,A -85,B 0,C 180,E1 -14174.362,E2 -14174.362} C_VEL
LIN {X 0,Y 341.384,Z 268.315,A -85,B 0,C 180,E1 -14177.826,E2 -14177.826} C_VEL
LIN {X 0,Y 341.119,Z 266.399,A -85,B 0,C 180,E1 -14180.3,E2 -14180.3} C_VEL
LIN {X 0,Y 340.802,Z 264.036,A -85,B 0,C 180,E1 -14183.536,E2 -14183.536} C_VEL
LIN {X 0,Y 340.727,Z 263.548,A -85,B 0,C 180,E1 -14184.716,E2 -14184.716} C_VEL
LIN {X 0,Y 340.701,Z 263.544,A -85,B 0,C 180,E1 -14188.95,E2 -14188.95} C_VEL
LIN {X 0,Y 340.726,Z 263.54,A -85,B 0,C 180,E1 -14193.007,E2 -14193.007} C_VEL
LIN {X 0,Y 340.713,Z 263.542,A -85,B 0,C 180,E1 -14196.92,E2 -14196.92} C_VEL
LIN {X 0,Y 340.737,Z 263.538,A -85,B 0,C 180,E1 -14200.724,E2 -14200.724} C_VEL
LIN {X 0,Y 340.818,Z 263.528,A -85,B 0,C 180,E1 -14204.444,E2 -14204.444} C_VEL
LIN {X 0,Y 340.847,Z 263.526,A -85,B 0,C 180,E1 -14208.094,E2 -14208.094} C_VEL
LIN {X 0,Y 340.977,Z 263.512,A -85,B 0,C 180,E1 -14211.698,E2 -14211.698} C_VEL
LIN {X 0,Y 341.02,Z 263.503,A -85,B 0,C 180,E1 -14214.079,E2 -14214.079} C_VEL
LIN {X 0,Y 341.12,Z 263.493,A -85,B 0,C 180,E1 -14217.632,E2 -14217.632} C_VEL
LIN {X 0,Y 341.246,Z 263.473,A -85,B 0,C 180,E1 -14219.993,E2 -14219.993} C_VEL
LIN {X 0,Y 341.155,Z 263.483,A -85,B 0,C 180,E1 -14222.354,E2 -14222.354} C_VEL
LIN {X 0,Y 341.027,Z 263.508,A -85,B 0,C 180,E1 -14227.095,E2 -14227.095} C_VEL
LIN {X 0,Y 340.831,Z 263.529,A -85,B 0,C 180,E1 -14230.687,E2 -14230.687} C_VEL
LIN {X 0,Y 340.844,Z 263.526,A -85,B 0,C 180,E1 -14234.318,E2 -14234.318} C_VEL
LIN {X 0,Y 340.762,Z 263.538,A -85,B 0,C 180,E1 -14238.433,E2 -14238.433} C_VEL
LIN {X 0,Y 340.693,Z 263.544,A -85,B 0,C 180,E1 -14241.834,E2 -14241.834} C_VEL
LIN {X 0,Y 340.743,Z 263.537,A -85,B 0,C 180,E1 -14245.657,E2 -14245.657} C_VEL
LIN {X 0,Y 340.688,Z 263.548,A -85,B 0,C 180,E1 -14248.315,E2 -14248.315} C_VEL
LIN {X 0,Y 340.662,Z 263.549,A -85,B 0,C 180,E1 -14251.038,E2 -14251.038} C_VEL
LIN {X 0,Y 340.681,Z 263.545,A -85,B 0,C 180,E1 -14255.272,E2 -14255.272} C_VEL
LIN {X 0,Y 340.674,Z 263.551,A -85,B 0,C 180,E1 -14258.38,E2 -14258.38} C_VEL
LIN {X 0,Y 340.686,Z 263.545,A -85,B 0,C 180,E1 -14261.297,E2 -14261.297} C_VEL
LIN {X 0,Y 340.738,Z 263.54,A -85,B 0,C 180,E1 -14264.516,E2 -14264.516} C_VEL
LIN {X 0,Y 340.705,Z 263.547,A -85,B 0,C 180,E1 -14267.939,E2 -14267.939} C_VEL
LIN {X 0,Y 340.686,Z 263.548,A -85,B 0,C 180,E1 -14270.247,E2 -14270.247} C_VEL
LIN {X 0,Y 340.66,Z 263.551,A -85,B 0,C 180,E1 -14273.554,E2 -14273.554} C_VEL
LIN {X 0,Y 340.64,Z 263.553,A -85,B 0,C 180,E1 -14276.148,E2 -14276.148} C_VEL
LIN {X 0,Y 340.721,Z 263.542,A -85,B 0,C 180,E1 -14280.328,E2 -14280.328} C_VEL
LIN {X 0,Y 340.75,Z 263.538,A -85,B 0,C 180,E1 -14283.016,E2 -14283.016} C_VEL
LIN {X 0,Y 340.734,Z 263.54,A -85,B 0,C 180,E1 -14286.928,E2 -14286.928} C_VEL
LIN {X 0,Y 340.74,Z 263.543,A -85,B 0,C 180,E1 -14289.829,E2 -14289.829} C_VEL
LIN {X 0,Y 341.676,Z 266.275,A -85,B 0,C 180,E1 -14290.08,E2 -14290.08} C_VEL
LIN {X 0,Y 343.807,Z 268.552,A -85,B 0,C 180,E1 -14290.506,E2 -14290.506} C_VEL
LIN {X 0,Y 346.227,Z 272.186,A -85,B 0,C 180,E1 -14291.025,E2 -14291.025} C_VEL
LIN {X 0,Y 348.314,Z 274.416,A -85,B 0,C 180,E1 -14291.469,E2 -14291.469} C_VEL
LIN {X 0,Y 351.043,Z 277.974,A -85,B 0,C 180,E1 -14292.092,E2 -14292.092} C_VEL
LIN {X 0,Y 353.163,Z 280.108,A -85,B 0,C 180,E1 -14292.557,E2 -14292.557} C_VEL
LIN {X 0,Y 356.456,Z 283.971,A -85,B 0,C 180,E1 -14293.361,E2 -14293.361} C_VEL
LIN {X 0,Y 358.638,Z 286.026,A -85,B 0,C 180,E1 -14293.88,E2 -14293.88} C_VEL
LIN {X 0,Y 362.117,Z 289.86,A -85,B 0,C 180,E1 -14294.804,E2 -14294.804} C_VEL
LIN {X 0,Y 364.957,Z 292.308,A -85,B 0,C 180,E1 -14295.564,E2 -14295.564} C_VEL
LIN {X 0,Y 368.412,Z 295.988,A -85,B 0,C 180,E1 -14296.588,E2 -14296.588} C_VEL
LIN {X 0,Y 372.014,Z 298.888,A -85,B 0,C 180,E1 -14297.727,E2 -14297.727} C_VEL
LIN {X 0,Y 375.348,Z 302.383,A -85,B 0,C 180,E1 -14298.935,E2 -14298.935} C_VEL
LIN {X 0,Y 379.017,Z 305,A -85,B 0,C 180,E1 -14300.394,E2 -14300.394} C_VEL
LIN {X 0,Y 380.549,Z 306.027,A -85,B 0,C 180,E1 -14301.064,E2 -14301.064} C_VEL
LIN {X 0,Y 383.285,Z 309.18,A -85,B 0,C 180,E1 -14302.551,E2 -14302.551} C_VEL
LIN {X 0,Y 385.767,Z 311.167,A -85,B 0,C 180,E1 -14304.136,E2 -14304.136} C_VEL
LIN {X 0,Y 387.876,Z 312.252,A -85,B 0,C 180,E1 -14305.844,E2 -14305.844} C_VEL
LIN {X 0,Y 388.849,Z 312.493,A -85,B 0,C 180,E1 -14306.892,E2 -14306.892} C_VEL
LIN {X 0,Y 389.946,Z 312.719,A -85,B 0,C 180,E1 -14308.967,E2 -14308.967} C_VEL
LIN {X 0,Y 390.096,Z 312.746,A -85,B 0,C 180,E1 -14310,E2 -14310} C_VEL
LIN {X 0,Y 389.524,Z 312.663,A -85,B 0,C 180,E1 -14312.068,E2 -14312.068} C_VEL
LIN {X 0,Y 388.355,Z 312.404,A -85,B 0,C 180,E1 -14313.667,E2 -14313.667} C_VEL
LIN {X 0,Y 386.366,Z 311.55,A -85,B 0,C 180,E1 -14315.439,E2 -14315.439} C_VEL
LIN {X 0,Y 383.826,Z 309.684,A -85,B 0,C 180,E1 -14317.131,E2 -14317.131} C_VEL
LIN {X 0,Y 380.963,Z 306.591,A -85,B 0,C 180,E1 -14318.718,E2 -14318.718} C_VEL
LIN {X 0,Y 380.001,Z 305.474,A -85,B 0,C 180,E1 -14319.186,E2 -14319.186} C_VEL
LIN {X 0,Y 376.77,Z 303.549,A -85,B 0,C 180,E1 -14320.522,E2 -14320.522} C_VEL
LIN {X 0,Y 373.24,Z 300.277,A -85,B 0,C 180,E1 -14321.844,E2 -14321.844} C_VEL
LIN {X 0,Y 371.161,Z 298.064,A -85,B 0,C 180,E1 -14322.559,E2 -14322.559} C_VEL
LIN {X 0,Y 367.31,Z 295.012,A -85,B 0,C 180,E1 -14323.738,E2 -14323.738} C_VEL
LIN {X 0,Y 363.887,Z 291.255,A -85,B 0,C 180,E1 -14324.738,E2 -14324.738} C_VEL
LIN {X 0,Y 360.07,Z 287.835,A -85,B 0,C 180,E1 -14325.73,E2 -14325.73} C_VEL
LIN {X 0,Y 357.577,Z 284.873,A -85,B 0,C 180,E1 -14326.381,E2 -14326.381} C_VEL
LIN {X 0,Y 354.154,Z 281.478,A -85,B 0,C 180,E1 -14327.197,E2 -14327.197} C_VEL
LIN {X 0,Y 352.027,Z 278.872,A -85,B 0,C 180,E1 -14327.695,E2 -14327.695} C_VEL
LIN {X 0,Y 348.914,Z 275.382,A -85,B 0,C 180,E1 -14328.39,E2 -14328.39} C_VEL
LIN {X 0,Y 347.407,Z 273.342,A -85,B 0,C 180,E1 -14328.729,E2 -14328.729} C_VEL
LIN {X 0,Y 344.82,Z 270.295,A -85,B 0,C 180,E1 -14329.273,E2 -14329.273} C_VEL
LIN {X 0,Y 343.676,Z 268.431,A -85,B 0,C 180,E1 -14329.519,E2 -14329.519} C_VEL
LIN {X 0,Y 341.638,Z 266.208,A -85,B 0,C 180,E1 -14329.928,E2 -14329.928} C_VEL
LIN {X 0,Y 340.744,Z 263.542,A -85,B 0,C 180,E1 -14330.192,E2 -14330.192} C_VEL
LIN {X 0,Y 340.734,Z 263.54,A -85,B 0,C 180,E1 -14333.072,E2 -14333.072} C_VEL
LIN {X 0,Y 340.75,Z 263.538,A -85,B 0,C 180,E1 -14336.984,E2 -14336.984} C_VEL
LIN {X 0,Y 340.709,Z 263.545,A -85,B 0,C 180,E1 -14339.982,E2 -14339.982} C_VEL
LIN {X 0,Y 340.64,Z 263.553,A -85,B 0,C 180,E1 -14343.852,E2 -14343.852} C_VEL
LIN {X 0,Y 340.655,Z 263.549,A -85,B 0,C 180,E1 -14346.747,E2 -14346.747} C_VEL
LIN {X 0,Y 340.716,Z 263.544,A -85,B 0,C 180,E1 -14350.267,E2 -14350.267} C_VEL
LIN {X 0,Y 340.734,Z 263.543,A -85,B 0,C 180,E1 -14353.801,E2 -14353.801} C_VEL
LIN {X 0,Y 340.72,Z 263.541,A -85,B 0,C 180,E1 -14357.115,E2 -14357.115} C_VEL
LIN {X 0,Y 340.694,Z 263.545,A -85,B 0,C 180,E1 -14360.259,E2 -14360.259} C_VEL
LIN {X 0,Y 340.673,Z 263.551,A -85,B 0,C 180,E1 -14363.566,E2 -14363.566} C_VEL
LIN {X 0,Y 340.659,Z 263.549,A -85,B 0,C 180,E1 -14366.16,E2 -14366.16} C_VEL
LIN {X 0,Y 340.697,Z 263.543,A -85,B 0,C 180,E1 -14370.335,E2 -14370.335} C_VEL
LIN {X 0,Y 340.761,Z 263.537,A -85,B 0,C 180,E1 -14373.026,E2 -14373.026} C_VEL
LIN {X 0,Y 340.732,Z 263.539,A -85,B 0,C 180,E1 -14374.667,E2 -14374.667} C_VEL
LIN {X 0,Y 340.05,Z 263.628,A -85,B 0,C 180,E1 -14375.653,E2 -14375.653} C_VEL
LIN {X 0,Y 337.159,Z 263.989,A -85,B 0,C 180,E1 -14377.258,E2 -14377.258} C_VEL
LIN {X 0,Y 334.724,Z 264.288,A -85,B 0,C 180,E1 -14378.557,E2 -14378.557} C_VEL
LIN {X 0,Y 333.696,Z 264.417,A -85,B 0,C 180,E1 -14379.563,E2 -14379.563} C_VEL
LIN {X 0,Y 333.622,Z 264.423,A -85,B 0,C 180,E1 -14379.904,E2 -14379.904} C_VEL
LIN {X 0,Y 333.697,Z 264.418,A -85,B 0,C 180,E1 -14382.86,E2 -14382.86} C_VEL
LIN {X 0,Y 333.774,Z 264.407,A -85,B 0,C 180,E1 -14386.616,E2 -14386.616} C_VEL
LIN {X 0,Y 333.804,Z 264.402,A -85,B 0,C 180,E1 -14390.311,E2 -14390.311} C_VEL
LIN {X 0,Y 333.989,Z 264.379,A -85,B 0,C 180,E1 -14393.968,E2 -14393.968} C_VEL
LIN {X 0,Y 334.092,Z 264.362,A -85,B 0,C 180,E1 -14397.596,E2 -14397.596} C_VEL
LIN {X 0,Y 334.198,Z 264.351,A -85,B 0,C 180,E1 -14400.007,E2 -14400.007} C_VEL
LIN {X 0,Y 334.061,Z 264.372,A -85,B 0,C 180,E1 -14402.418,E2 -14402.418} C_VEL
LIN {X 0,Y 333.994,Z 264.379,A -85,B 0,C 180,E1 -14406.046,E2 -14406.046} C_VEL
LIN {X 0,Y 333.818,Z 264.401,A -85,B 0,C 180,E1 -14409.703,E2 -14409.703} C_VEL
LIN {X 0,Y 333.797,Z 264.403,A -85,B 0,C 180,E1 -14413.398,E2 -14413.398} C_VEL
LIN {X 0,Y 333.721,Z 264.413,A -85,B 0,C 180,E1 -14417.154,E2 -14417.154} C_VEL
LIN {X 0,Y 333.674,Z 264.419,A -85,B 0,C 180,E1 -14419.7,E2 -14419.7} C_VEL
LIN {X 0,Y 333.654,Z 264.422,A -85,B 0,C 180,E1 -14423.597,E2 -14423.597} C_VEL
LIN {X 0,Y 333.643,Z 264.427,A -85,B 0,C 180,E1 -14426.26,E2 -14426.26} C_VEL
LIN {X 0,Y 333.661,Z 264.42,A -85,B 0,C 180,E1 -14428.983,E2 -14428.983} C_VEL
LIN {X 0,Y 333.653,Z 264.424,A -85,B 0,C 180,E1 -14432.592,E2 -14432.592} C_VEL
LIN {X 0,Y 333.694,Z 264.42,A -85,B 0,C 180,E1 -14434.778,E2 -14434.778} C_VEL
LIN {X 0,Y 333.808,Z 265.441,A -85,B 0,C 180,E1 -14436.867,E2 -14436.867} C_VEL
LIN {X 0,Y 334.224,Z 268.35,A -85,B 0,C 180,E1 -14440.801,E2 -14440.801} C_VEL
LIN {X 0,Y 334.605,Z 271.252,A -85,B 0,C 180,E1 -14444.429,E2 -14444.429} C_VEL
LIN {X 0,Y 334.719,Z 274.239,A -85,B 0,C 180,E1 -14447.788,E2 -14447.788} C_VEL
LIN {X 0,Y 334.417,Z 277.385,A -85,B 0,C 180,E1 -14451.046,E2 -14451.046} C_VEL
LIN {X 0,Y 334.058,Z 280.309,A -85,B 0,C 180,E1 -14453.91,E2 -14453.91} C_VEL
LIN {X 0,Y 333.57,Z 284.097,A -85,B 0,C 180,E1 -14457.44,E2 -14457.44} C_VEL
LIN {X 0,Y 333.042,Z 288.072,A -85,B 0,C 180,E1 -14460.965,E2 -14460.965} C_VEL
LIN {X 0,Y 332.648,Z 292.782,A -85,B 0,C 180,E1 -14465.005,E2 -14465.005} C_VEL
LIN {X 0,Y 332.393,Z 296.672,A -85,B 0,C 180,E1 -14468.171,E2 -14468.171} C_VEL
LIN {X 0,Y 334.732,Z 306.696,A -85,B 0,C 180,E1 -14468.723,E2 -14468.723} C_VEL
LIN {X 0,Y 336.823,Z 317.432,A -85,B 0,C 180,E1 -14469.451,E2 -14469.451} C_VEL
LIN {X 0,Y 338.409,Z 328.657,A -85,B 0,C 180,E1 -14470.366,E2 -14470.366} C_VEL
LIN {X 0,Y 339.133,Z 336.316,A -85,B 0,C 180,E1 -14471.107,E2 -14471.107} C_VEL
LIN {X 0,Y 338.23,Z 345.033,A -85,B 0,C 180,E1 -14471.996,E2 -14471.996} C_VEL
LIN {X 0,Y 337.093,Z 353.541,A -85,B 0,C 180,E1 -14473.03,E2 -14473.03} C_VEL
LIN {X 0,Y 336.14,Z 361.723,A -85,B 0,C 180,E1 -14474.229,E2 -14474.229} C_VEL
LIN {X 0,Y 335.075,Z 370.278,A -85,B 0,C 180,E1 -14475.733,E2 -14475.733} C_VEL
LIN {X 0,Y 333.925,Z 378.606,A -85,B 0,C 180,E1 -14477.542,E2 -14477.542} C_VEL
LIN {X 0,Y 333.248,Z 384.265,A -85,B 0,C 180,E1 -14479.059,E2 -14479.059} C_VEL
LIN {X 0,Y 332.6,Z 389.757,A -85,B 0,C 180,E1 -14480.882,E2 -14480.882} C_VEL
LIN {X 0,Y 332.218,Z 394.083,A -85,B 0,C 180,E1 -14482.708,E2 -14482.708} C_VEL
LIN {X 0,Y 332.049,Z 396.827,A -85,B 0,C 180,E1 -14484.179,E2 -14484.179} C_VEL
LIN {X 0,Y 331.973,Z 399.64,A -85,B 0,C 180,E1 -14486.359,E2 -14486.359} C_VEL
LIN {X 0,Y 331.921,Z 400.698,A -85,B 0,C 180,E1 -14487.573,E2 -14487.573} C_VEL
LIN {X 0,Y 331.912,Z 401.287,A -85,B 0,C 180,E1 -14488.787,E2 -14488.787} C_VEL
LIN {X 0,Y 331.912,Z 401.287,A -85,B 0,C 180,E1 -14491.213,E2 -14491.213} C_VEL
LIN {X 0,Y 331.921,Z 400.698,A -85,B 0,C 180,E1 -14492.427,E2 -14492.427} C_VEL
LIN {X 0,Y 331.978,Z 398.251,A -85,B 0,C 180,E1 -14494.858,E2 -14494.858} C_VEL
LIN {X 0,Y 332.126,Z 395.3,A -85,B 0,C 180,E1 -14496.683,E2 -14496.683} C_VEL
LIN {X 0,Y 332.471,Z 391.312,A -85,B 0,C 180,E1 -14498.509,E2 -14498.509} C_VEL
LIN {X 0,Y 332.997,Z 386.181,A -85,B 0,C 180,E1 -14500.334,E2 -14500.334} C_VEL
LIN {X 0,Y 333.606,Z 380.918,A -85,B 0,C 180,E1 -14501.853,E2 -14501.853} C_VEL
LIN {X 0,Y 334.484,Z 374.602,A -85,B 0,C 180,E1 -14503.363,E2 -14503.363} C_VEL
LIN {X 0,Y 335.24,Z 368.65,A -85,B 0,C 180,E1 -14504.57,E2 -14504.57} C_VEL
LIN {X 0,Y 336.251,Z 360.598,A -85,B 0,C 180,E1 -14505.948,E2 -14505.948} C_VEL
LIN {X 0,Y 337.21,Z 352.405,A -85,B 0,C 180,E1 -14507.12,E2 -14507.12} C_VEL
LIN {X 0,Y 338.325,Z 343.68,A -85,B 0,C 180,E1 -14508.155,E2 -14508.155} C_VEL
LIN {X 0,Y 339.091,Z 336.314,A -85,B 0,C 180,E1 -14508.895,E2 -14508.895} C_VEL
LIN {X 0,Y 338.185,Z 326.836,A -85,B 0,C 180,E1 -14509.789,E2 -14509.789} C_VEL
LIN {X 0,Y 336.826,Z 317.432,A -85,B 0,C 180,E1 -14510.549,E2 -14510.549} C_VEL
LIN {X 0,Y 334.853,Z 307.145,A -85,B 0,C 180,E1 -14511.248,E2 -14511.248} C_VEL
LIN {X 0,Y 332.493,Z 297.603,A -85,B 0,C 180,E1 -14511.794,E2 -14511.794} C_VEL
LIN {X 0,Y 332.369,Z 296.529,A -85,B 0,C 180,E1 -14511.862,E2 -14511.862} C_VEL
LIN {X 0,Y 332.646,Z 292.772,A -85,B 0,C 180,E1 -14514.995,E2 -14514.995} C_VEL
LIN {X 0,Y 333.039,Z 288.047,A -85,B 0,C 180,E1 -14519.035,E2 -14519.035} C_VEL
LIN {X 0,Y 333.574,Z 284.094,A -85,B 0,C 180,E1 -14522.561,E2 -14522.561} C_VEL
LIN {X 0,Y 334.06,Z 280.301,A -85,B 0,C 180,E1 -14526.09,E2 -14526.09} C_VEL
LIN {X 0,Y 334.426,Z 277.247,A -85,B 0,C 180,E1 -14529.082,E2 -14529.082} C_VEL
LIN {X 0,Y 334.694,Z 274.213,A -85,B 0,C 180,E1 -14532.216,E2 -14532.216} C_VEL
LIN {X 0,Y 334.704,Z 272.196,A -85,B 0,C 180,E1 -14534.439,E2 -14534.439} C_VEL
LIN {X 0,Y 334.368,Z 269.429,A -85,B 0,C 180,E1 -14537.726,E2 -14537.726} C_VEL
LIN {X 0,Y 334.009,Z 266.867,A -85,B 0,C 180,E1 -14541.124,E2 -14541.124} C_VEL
LIN {X 0,Y 333.767,Z 264.939,A -85,B 0,C 180,E1 -14543.866,E2 -14543.866} C_VEL
LIN {X 0,Y 333.684,Z 264.426,A -85,B 0,C 180,E1 -14545.336,E2 -14545.336} C_VEL
LIN {X 0,Y 333.638,Z 264.428,A -85,B 0,C 180,E1 -14548.217,E2 -14548.217} C_VEL
LIN {X 0,Y 333.661,Z 264.421,A -85,B 0,C 180,E1 -14551.017,E2 -14551.017} C_VEL
LIN {X 0,Y 333.677,Z 264.419,A -85,B 0,C 180,E1 -14555.081,E2 -14555.081} C_VEL
LIN {X 0,Y 333.667,Z 264.42,A -85,B 0,C 180,E1 -14559.012,E2 -14559.012} C_VEL
LIN {X 0,Y 333.744,Z 264.415,A -85,B 0,C 180,E1 -14561.58,E2 -14561.58} C_VEL
LIN {X 0,Y 333.81,Z 264.407,A -85,B 0,C 180,E1 -14565.571,E2 -14565.571} C_VEL
LIN {X 0,Y 333.815,Z 264.403,A -85,B 0,C 180,E1 -14569.071,E2 -14569.071} C_VEL
LIN {X 0,Y 333.967,Z 264.382,A -85,B 0,C 180,E1 -14572.74,E2 -14572.74} C_VEL
LIN {X 0,Y 333.783,Z 264.408,A -85,B 0,C 180,E1 -14575.162,E2 -14575.162} C_VEL
LIN {X 0,Y 334.061,Z 264.372,A -85,B 0,C 180,E1 -14577.582,E2 -14577.582} C_VEL
LIN {X 0,Y 334.198,Z 264.351,A -85,B 0,C 180,E1 -14579.993,E2 -14579.993} C_VEL
LIN {X 0,Y 334.092,Z 264.362,A -85,B 0,C 180,E1 -14582.404,E2 -14582.404} C_VEL
LIN {X 0,Y 333.964,Z 264.381,A -85,B 0,C 180,E1 -14586.594,E2 -14586.594} C_VEL
LIN {X 0,Y 333.804,Z 264.402,A -85,B 0,C 180,E1 -14589.689,E2 -14589.689} C_VEL
LIN {X 0,Y 333.774,Z 264.407,A -85,B 0,C 180,E1 -14593.384,E2 -14593.384} C_VEL
LIN {X 0,Y 333.697,Z 264.418,A -85,B 0,C 180,E1 -14597.14,E2 -14597.14} C_VEL
LIN {X 0,Y 333.64,Z 264.421,A -85,B 0,C 180,E1 -14599.687,E2 -14599.687} C_VEL
LIN {X 0,Y 333.642,Z 264.422,A -85,B 0,C 180,E1 -14603.583,E2 -14603.583} C_VEL
LIN {X 0,Y 333.7,Z 264.417,A -85,B 0,C 180,E1 -14606.24,E2 -14606.24} C_VEL
LIN {X 0,Y 333.649,Z 264.423,A -85,B 0,C 180,E1 -14608.968,E2 -14608.968} C_VEL
LIN {X 0,Y 333.604,Z 264.427,A -85,B 0,C 180,E1 -14613.201,E2 -14613.201} C_VEL
LIN {X 0,Y 333.628,Z 264.425,A -85,B 0,C 180,E1 -14616.825,E2 -14616.825} C_VEL
LIN {X 0,Y 333.659,Z 264.421,A -85,B 0,C 180,E1 -14620.753,E2 -14620.753} C_VEL
LIN {X 0,Y 333.687,Z 264.421,A -85,B 0,C 180,E1 -14624.268,E2 -14624.268} C_VEL
LIN {X 0,Y 333.66,Z 264.422,A -85,B 0,C 180,E1 -14627.623,E2 -14627.623} C_VEL
LIN {X 0,Y 333.631,Z 264.424,A -85,B 0,C 180,E1 -14631.191,E2 -14631.191} C_VEL
